C03648=1017.335,-79.595,386.221,-24.023,21.641,-43.975
C03649=1017.333,-79.935,386.245,-24.022,21.641,-43.981
C03650=1017.331,-80.274,386.270,-24.021,21.641,-43.986
C03651=1017.330,-80.613,386.294,-24.021,21.643,-43.990
C03652=1017.328,-80.952,386.319,-24.020,21.643,-43.995
C03653=1017.326,-81.290,386.344,-24.020,21.643,-44.001
C03654=1017.325,-81.627,386.368,-24.019,21.644,-44.005
C03655=1017.323,-81.965,386.392,-24.018,21.645,-44.010
C03656=1017.321,-82.302,386.417,-24.018,21.645,-44.016
C03657=1017.319,-82.639,386.441,-24.017,21.645,-44.021
C03658=1017.317,-82.974,386.465,-24.016,21.646,-44.025
C03659=1017.315,-83.310,386.490,-24.016,21.647,-44.031
C03660=1017.313,-83.646,386.514,-24.015,21.647,-44.036
C03661=1017.312,-83.981,386.538,-24.015,21.648,-44.040
C03662=1017.310,-84.315,386.562,-24.014,21.648,-44.045
C03663=1017.307,-84.664,386.587,-24.013,21.649,-44.051
C03664=1017.305,-85.062,386.616,-24.012,21.650,-44.056
C03665=1017.304,-85.273,386.631,-24.012,21.649,-44.060
C03666=1017.303,-85.488,386.647,-24.012,21.649,-44.062
C03667=1017.301,-85.897,386.676,-24.011,21.650,-44.067
C03668=1017.299,-86.255,386.702,-24.010,21.651,-44.073
C03669=1017.296,-86.585,386.726,-24.009,21.652,-44.078
C03670=1017.294,-86.907,386.749,-24.009,21.652,-44.082
C03671=1017.292,-87.224,386.772,-24.008,21.653,-44.088
C03672=1017.290,-87.536,386.794,-24.007,21.653,-44.093
C03673=1017.288,-87.847,386.816,-24.007,21.654,-44.097
C03674=1017.286,-88.160,386.839,-24.006,21.654,-44.102
C03675=1017.284,-88.478,386.861,-24.006,21.655,-44.106
C03676=1017.283,-88.849,386.888,-24.005,21.656,-44.114
C03677=1017.281,-89.068,386.904,-24.004,21.656,-44.117
C03678=1017.279,-89.302,386.921,-24.004,21.656,-44.119
C03679=1017.278,-89.540,386.938,-24.004,21.656,-44.121
C03680=1017.277,-89.771,386.954,-24.004,21.657,-44.123
C03681=1017.273,-90.177,386.983,-24.003,21.658,-44.130
C03682=1017.271,-90.516,387.008,-24.002,21.658,-44.136
C03683=1017.269,-90.845,387.031,-24.001,21.659,-44.141
C03684=1017.267,-91.173,387.055,-24.001,21.660,-44.145
C03685=1017.264,-91.502,387.078,-24.000,21.660,-44.150
C03686=1017.262,-91.831,387.101,-23.999,21.660,-44.156
C03687=1017.260,-92.159,387.125,-23.999,21.661,-44.160
C03688=1017.258,-92.486,387.148,-23.998,21.662,-44.165
C03689=1017.256,-92.813,387.171,-23.998,21.662,-44.169
C03690=1017.253,-93.139,387.194,-23.997,21.663,-44.175
C03691=1017.251,-93.465,387.218,-23.996,21.663,-44.180
C03692=1017.248,-93.789,387.240,-23.996,21.664,-44.184
C03693=1017.246,-94.114,387.264,-23.995,21.664,-44.189
C03694=1017.243,-94.438,387.287,-23.994,21.665,-44.193
C03695=1017.241,-94.762,387.310,-23.994,21.666,-44.199
C03696=1017.239,-95.085,387.333,-23.993,21.666,-44.204
C03697=1017.237,-95.407,387.356,-23.993,21.666,-44.207
C03698=1017.234,-95.729,387.378,-23.992,21.667,-44.213
C03699=1017.232,-96.052,387.402,-23.991,21.668,-44.217
C03700=1017.229,-96.373,387.424,-23.991,21.668,-44.222
C03701=1017.226,-96.695,387.447,-23.990,21.669,-44.226
C03702=1017.224,-97.016,387.469,-23.989,21.669,-44.231
C03703=1017.222,-97.337,387.492,-23.989,21.670,-44.236
C03704=1017.219,-97.658,387.515,-23.988,21.670,-44.241
C03705=1017.216,-97.979,387.538,-23.987,21.670,-44.246
C03706=1017.214,-98.300,387.560,-23.987,21.672,-44.250
C03707=1017.212,-98.620,387.583,-23.986,21.671,-44.255
C03708=1017.209,-98.942,387.605,-23.986,21.673,-44.260
C03709=1017.207,-99.263,387.628,-23.985,21.673,-44.265
C03710=1017.204,-99.585,387.651,-23.985,21.673,-44.268
C03711=1017.202,-99.906,387.673,-23.984,21.674,-44.274
C03712=1017.199,-100.227,387.696,-23.983,21.675,-44.278
C03713=1017.196,-100.551,387.719,-23.983,21.675,-44.283
C03714=1017.194,-100.872,387.742,-23.982,21.676,-44.287
C03715=1017.190,-101.196,387.764,-23.981,21.676,-44.292
C03716=1017.188,-101.519,387.786,-23.981,21.677,-44.298
C03717=1017.185,-101.843,387.810,-23.980,21.677,-44.302
C03718=1017.182,-102.168,387.833,-23.980,21.678,-44.307
C03719=1017.180,-102.493,387.855,-23.979,21.679,-44.311
C03720=1017.177,-102.818,387.878,-23.978,21.679,-44.316
C03721=1017.174,-103.145,387.901,-23.978,21.680,-44.320
C03722=1017.171,-103.471,387.924,-23.977,21.680,-44.326
C03723=1017.168,-103.798,387.947,-23.976,21.681,-44.331
C03724=1017.165,-104.125,387.970,-23.976,21.681,-44.335
C03725=1017.163,-104.453,387.992,-23.975,21.681,-44.340
C03726=1017.159,-104.781,388.016,-23.975,21.683,-44.344
C03727=1017.156,-105.110,388.038,-23.974,21.683,-44.350
C03728=1017.153,-105.438,388.061,-23.974,21.684,-44.354
C03729=1017.151,-105.767,388.084,-23.973,21.684,-44.359
C03730=1017.148,-106.096,388.107,-23.972,21.685,-44.365
C03731=1017.144,-106.425,388.130,-23.972,21.685,-44.368
C03732=1017.141,-106.754,388.153,-23.971,21.685,-44.374
C03733=1017.139,-107.083,388.176,-23.971,21.687,-44.378
C03734=1017.135,-107.412,388.199,-23.970,21.687,-44.383
C03735=1017.132,-107.740,388.222,-23.969,21.687,-44.388
C03736=1017.129,-108.070,388.245,-23.969,21.688,-44.392
C03737=1017.126,-108.398,388.268,-23.968,21.689,-44.398
C03738=1017.122,-108.727,388.291,-23.967,21.689,-44.402
C03739=1017.120,-109.056,388.314,-23.967,21.689,-44.407
C03740=1017.117,-109.385,388.337,-23.966,21.690,-44.412
C03741=1017.113,-109.714,388.360,-23.965,21.691,-44.416
C03742=1017.110,-110.043,388.382,-23.965,21.691,-44.422
C03743=1017.107,-110.372,388.404,-23.964,21.692,-44.426
C03744=1017.104,-110.701,388.427,-23.963,21.692,-44.431
C03745=1017.101,-111.030,388.450,-23.963,21.693,-44.436
C03746=1017.096,-111.359,388.473,-23.962,21.693,-44.440
C03747=1017.093,-111.687,388.495,-23.962,21.694,-44.446
C03748=1017.090,-112.016,388.518,-23.961,21.695,-44.449
C03749=1017.087,-112.345,388.541,-23.960,21.695,-44.455
C03750=1017.084,-112.674,388.564,-23.960,21.696,-44.459
C03751=1017.080,-113.002,388.587,-23.959,21.696,-44.464
C03752=1017.076,-113.330,388.609,-23.958,21.697,-44.470
C03753=1017.073,-113.659,388.632,-23.958,21.697,-44.473
C03754=1017.070,-113.988,388.655,-23.957,21.698,-44.479
C03755=1017.066,-114.316,388.677,-23.957,21.699,-44.483
C03756=1017.062,-114.645,388.700,-23.956,21.699,-44.488
C03757=1017.059,-114.974,388.723,-23.956,21.700,-44.492
C03758=1017.056,-115.302,388.745,-23.955,21.700,-44.497
C03759=1017.053,-115.631,388.768,-23.954,21.701,-44.503
C03760=1017.048,-115.960,388.790,-23.954,21.701,-44.507
C03761=1017.045,-116.288,388.813,-23.953,21.701,-44.512
C03762=1017.041,-116.616,388.836,-23.953,21.703,-44.516
C03763=1017.038,-116.945,388.858,-23.952,21.703,-44.521
C03764=1017.034,-117.273,388.881,-23.951,21.704,-44.525
C03765=1017.031,-117.602,388.904,-23.951,21.704,-44.531
C03766=1017.027,-117.930,388.926,-23.950,21.705,-44.535
C03767=1017.023,-118.259,388.948,-23.949,21.705,-44.540
C03768=1017.019,-118.588,388.971,-23.949,21.705,-44.545
C03769=1017.015,-118.915,388.994,-23.948,21.707,-44.549
C03770=1017.012,-119.244,389.016,-23.948,21.707,-44.554
C03771=1017.009,-119.572,389.038,-23.947,21.707,-44.558
C03772=1017.004,-119.901,389.061,-23.946,21.708,-44.564
C03773=1017.000,-120.229,389.083,-23.946,21.709,-44.568
C03774=1016.996,-120.557,389.106,-23.945,21.709,-44.573
C03775=1016.993,-120.885,389.128,-23.945,21.710,-44.577
C03776=1016.989,-121.214,389.150,-23.944,21.710,-44.582
C03777=1016.985,-121.543,389.173,-23.944,21.711,-44.586
C03778=1016.981,-121.871,389.196,-23.943,21.711,-44.591
C03779=1016.977,-122.199,389.218,-23.942,21.712,-44.597
C03780=1016.974,-122.510,389.239,-23.942,21.713,-44.601
C03781=1016.969,-122.856,389.263,-23.941,21.713,-44.606
C03782=1016.965,-123.184,389.285,-23.940,21.714,-44.610
C03783=1016.961,-123.512,389.308,-23.940,21.714,-44.615
C03784=1016.957,-123.840,389.330,-23.939,21.715,-44.620
C03785=1016.954,-124.168,389.352,-23.939,21.715,-44.625
C03786=1016.948,-124.496,389.374,-23.938,21.716,-44.628
C03787=1016.945,-124.825,389.396,-23.937,21.717,-44.634
C03788=1016.941,-125.153,389.419,-23.937,21.717,-44.638
C03789=1016.937,-125.481,389.441,-23.936,21.717,-44.643
C03790=1016.933,-125.809,389.463,-23.936,21.719,-44.647
C03791=1016.929,-126.138,389.486,-23.935,21.719,-44.652
C03792=1016.924,-126.466,389.507,-23.935,21.720,-44.657
C03793=1016.920,-126.793,389.530,-23.934,21.720,-44.662
C03794=1016.916,-127.122,389.552,-23.933,21.720,-44.667
C03795=1016.911,-127.450,389.574,-23.933,21.721,-44.671
C03796=1016.907,-127.778,389.597,-23.932,21.721,-44.676
C03797=1016.903,-128.106,389.619,-23.931,21.722,-44.680
C03798=1016.899,-128.434,389.641,-23.931,21.723,-44.686
C03799=1016.894,-128.762,389.664,-23.930,21.723,-44.689
C03800=1016.889,-129.090,389.685,-23.929,21.723,-44.695
C03801=1016.886,-129.419,389.707,-23.929,21.725,-44.699
C03802=1016.881,-129.746,389.730,-23.928,21.724,-44.704
C03803=1016.876,-130.075,389.752,-23.928,21.726,-44.708
C03804=1016.872,-130.403,389.774,-23.927,21.726,-44.713
C03805=1016.868,-130.730,389.796,-23.927,21.726,-44.717
C03806=1016.863,-131.058,389.818,-23.926,21.727,-44.723
C03807=1016.859,-131.387,389.840,-23.926,21.728,-44.726
C03808=1016.854,-131.715,389.863,-23.925,21.728,-44.732
C03809=1016.850,-132.043,389.884,-23.924,21.729,-44.736
C03810=1016.846,-132.370,389.907,-23.924,21.729,-44.741
C03811=1016.840,-132.699,389.929,-23.923,21.730,-44.745
C03812=1016.836,-133.027,389.950,-23.922,21.731,-44.750
C03813=1016.832,-133.354,389.973,-23.922,21.731,-44.754
C03814=1016.827,-133.683,389.995,-23.921,21.731,-44.759
C03815=1016.822,-134.010,390.017,-23.921,21.732,-44.763
C03816=1017.213,-133.983,389.773,-23.921,21.732,-44.763
C03817=1017.218,-133.655,389.751,-23.921,21.731,-44.759
C03818=1017.222,-133.327,389.730,-23.922,21.731,-44.754
C03819=1017.227,-132.998,389.706,-23.922,21.731,-44.750
C03820=1017.232,-132.670,389.685,-23.923,21.730,-44.745
C03821=1017.236,-132.342,389.663,-23.924,21.729,-44.741
C03822=1017.240,-132.014,389.641,-23.924,21.729,-44.736
C03823=1017.245,-131.687,389.619,-23.925,21.728,-44.732
C03824=1017.250,-131.358,389.597,-23.926,21.728,-44.726
C03825=1017.254,-131.030,389.575,-23.926,21.727,-44.723
C03826=1017.258,-130.703,389.553,-23.927,21.726,-44.717
C03827=1017.262,-130.374,389.531,-23.927,21.726,-44.713
C03828=1017.267,-130.047,389.509,-23.928,21.726,-44.708
C03829=1017.270,-129.718,389.487,-23.928,21.724,-44.704
C03830=1017.275,-129.391,389.465,-23.929,21.725,-44.699
C03831=1017.280,-129.062,389.442,-23.929,21.723,-44.695
C03832=1017.283,-128.734,389.420,-23.930,21.723,-44.689
C03833=1017.288,-128.406,389.399,-23.931,21.723,-44.686
C03834=1017.292,-128.078,389.376,-23.931,21.722,-44.680
C03835=1017.296,-127.750,389.354,-23.932,21.721,-44.676
C03836=1017.300,-127.422,389.332,-23.933,21.721,-44.671
C03837=1017.304,-127.094,389.310,-23.933,21.720,-44.667
C03838=1017.308,-126.766,389.287,-23.934,21.720,-44.662
C03839=1017.313,-126.437,389.265,-23.935,21.720,-44.657
C03840=1017.317,-126.109,389.243,-23.935,21.719,-44.652
C03841=1017.321,-125.781,389.221,-23.936,21.719,-44.647
C03842=1017.325,-125.453,389.199,-23.936,21.717,-44.643
C03843=1017.329,-125.125,389.176,-23.937,21.717,-44.638
C03844=1017.332,-124.797,389.154,-23.937,21.717,-44.634
C03845=1017.336,-124.469,389.132,-23.938,21.716,-44.628
C03846=1017.340,-124.140,389.110,-23.939,21.715,-44.625
C03847=1017.345,-123.812,389.088,-23.939,21.715,-44.620
C03848=1017.349,-123.484,389.065,-23.940,21.714,-44.615
C03849=1017.353,-123.156,389.043,-23.940,21.714,-44.610
C03850=1017.357,-122.828,389.021,-23.941,21.713,-44.606
C03851=1017.360,-122.499,388.999,-23.942,21.713,-44.601
C03852=1017.364,-122.171,388.976,-23.942,21.712,-44.597
C03853=1017.367,-121.842,388.954,-23.943,21.711,-44.591
C03854=1017.371,-121.515,388.932,-23.944,21.711,-44.586
C03855=1017.376,-121.186,388.909,-23.944,21.710,-44.582
C03856=1017.380,-120.858,388.887,-23.945,21.710,-44.577
C03857=1017.383,-120.529,388.865,-23.945,21.709,-44.573
C03858=1017.386,-120.201,388.842,-23.946,21.709,-44.568
C03859=1017.390,-119.873,388.820,-23.946,21.708,-44.564
C03860=1017.394,-119.544,388.798,-23.947,21.707,-44.558
C03861=1017.398,-119.217,388.775,-23.948,21.707,-44.554
C03862=1017.402,-118.887,388.752,-23.948,21.707,-44.549
C03863=1017.405,-118.559,388.730,-23.949,21.705,-44.545
C03864=1017.409,-118.231,388.708,-23.949,21.705,-44.540
C03865=1017.412,-117.902,388.685,-23.950,21.705,-44.535
C03866=1017.416,-117.574,388.663,-23.951,21.704,-44.531
C03867=1017.419,-117.245,388.640,-23.951,21.704,-44.525
C03868=1017.423,-116.917,388.618,-23.952,21.703,-44.521
C03869=1017.426,-116.588,388.595,-23.953,21.703,-44.516
C03870=1017.430,-116.260,388.573,-23.953,21.701,-44.512
C03871=1017.433,-115.931,388.550,-23.954,21.701,-44.507
C03872=1017.437,-115.603,388.528,-23.954,21.701,-44.503
C03873=1017.440,-115.275,388.505,-23.955,21.700,-44.497
C03874=1017.444,-114.947,388.483,-23.956,21.700,-44.492
C03875=1017.448,-114.617,388.460,-23.956,21.699,-44.488
C03876=1017.451,-114.289,388.437,-23.957,21.699,-44.483
C03877=1017.455,-113.961,388.415,-23.957,21.698,-44.479
C03878=1017.458,-113.632,388.392,-23.958,21.697,-44.473
C03879=1017.461,-113.303,388.369,-23.958,21.697,-44.470
C03880=1017.464,-112.974,388.347,-23.959,21.696,-44.464
C03881=1017.467,-112.646,388.324,-23.960,21.696,-44.459
C03882=1017.471,-112.317,388.302,-23.960,21.695,-44.455
C03883=1017.474,-111.989,388.279,-23.961,21.695,-44.449
C03884=1017.477,-111.659,388.257,-23.962,21.694,-44.446
C03885=1017.480,-111.330,388.234,-23.962,21.693,-44.440
C03886=1017.484,-111.002,388.211,-23.963,21.693,-44.436
C03887=1017.487,-110.672,388.188,-23.963,21.692,-44.431
C03888=1017.490,-110.344,388.166,-23.964,21.692,-44.426
C03889=1017.493,-110.015,388.143,-23.965,21.691,-44.422
C03890=1017.496,-109.687,388.120,-23.965,21.691,-44.416
C03891=1017.500,-109.357,388.097,-23.966,21.690,-44.412
C03892=1017.503,-109.029,388.074,-23.967,21.689,-44.407
C03893=1017.506,-108.700,388.052,-23.967,21.689,-44.402
C03894=1017.510,-108.371,388.029,-23.968,21.689,-44.398
C03895=1017.512,-108.042,388.006,-23.969,21.688,-44.392
C03896=1017.515,-107.713,387.983,-23.969,21.687,-44.388
C03897=1017.518,-107.384,387.960,-23.970,21.687,-44.383
C03898=1017.521,-107.055,387.938,-23.971,21.687,-44.378
C03899=1017.524,-106.725,387.914,-23.971,21.685,-44.374
C03900=1017.527,-106.397,387.891,-23.972,21.685,-44.368
C03901=1017.530,-106.068,387.869,-23.972,21.685,-44.365
C03902=1017.533,-105.739,387.847,-23.973,21.684,-44.359
C03903=1017.536,-105.410,387.823,-23.974,21.684,-44.354
C03904=1017.539,-105.082,387.800,-23.974,21.683,-44.350
C03905=1017.542,-104.754,387.777,-23.975,21.683,-44.344
C03906=1017.545,-104.425,387.754,-23.975,21.681,-44.340
C03907=1017.547,-104.098,387.731,-23.976,21.681,-44.335
C03908=1017.550,-103.771,387.708,-23.976,21.681,-44.331
C03909=1017.553,-103.444,387.685,-23.977,21.680,-44.326
C03910=1017.556,-103.117,387.663,-23.978,21.680,-44.320
C03911=1017.558,-102.791,387.640,-23.978,21.679,-44.316
C03912=1017.561,-102.466,387.617,-23.979,21.679,-44.311
C03913=1017.565,-102.140,387.594,-23.980,21.678,-44.307
C03914=1017.567,-101.815,387.572,-23.980,21.677,-44.302
C03915=1017.570,-101.492,387.549,-23.981,21.677,-44.298
C03916=1017.572,-101.168,387.526,-23.981,21.676,-44.292
C03917=1017.575,-100.845,387.504,-23.982,21.676,-44.287
C03918=1017.577,-100.522,387.481,-23.983,21.675,-44.283
C03919=1017.580,-100.200,387.459,-23.983,21.675,-44.278
C03920=1017.583,-99.878,387.436,-23.984,21.674,-44.274
C03921=1017.586,-99.557,387.413,-23.985,21.673,-44.268
C03922=1017.588,-99.235,387.391,-23.985,21.673,-44.265
C03923=1017.590,-98.914,387.369,-23.986,21.673,-44.260
C03924=1017.593,-98.593,387.345,-23.986,21.671,-44.255
C03925=1017.595,-98.272,387.323,-23.987,21.672,-44.250
C03926=1017.598,-97.951,387.300,-23.987,21.670,-44.246
C03927=1017.600,-97.631,387.277,-23.988,21.670,-44.241
C03928=1017.602,-97.310,387.255,-23.989,21.670,-44.236
C03929=1017.605,-96.988,387.232,-23.989,21.669,-44.231
C03930=1017.607,-96.667,387.210,-23.990,21.669,-44.226
C03931=1017.610,-96.347,387.187,-23.991,21.668,-44.222
C03932=1017.612,-96.025,387.164,-23.991,21.668,-44.217
C03933=1017.615,-95.703,387.141,-23.992,21.667,-44.213
C03934=1017.617,-95.381,387.118,-23.993,21.666,-44.207
C03935=1017.620,-95.057,387.096,-23.993,21.666,-44.204
C03936=1017.622,-94.735,387.073,-23.994,21.666,-44.199
C03937=1017.624,-94.412,387.050,-23.994,21.665,-44.193
C03938=1017.626,-94.086,387.027,-23.995,21.664,-44.189
C03939=1017.629,-93.762,387.004,-23.996,21.664,-44.184
C03940=1017.631,-93.437,386.981,-23.996,21.663,-44.180
C03941=1017.633,-93.111,386.958,-23.997,21.663,-44.175
C03942=1017.636,-92.785,386.934,-23.998,21.662,-44.169
C03943=1017.638,-92.459,386.911,-23.998,21.662,-44.165
C03944=1017.640,-92.131,386.888,-23.999,21.661,-44.160
C03945=1017.642,-91.804,386.864,-23.999,21.660,-44.156
C03946=1017.645,-91.475,386.841,-24.000,21.660,-44.150
C03947=1017.646,-91.147,386.818,-24.001,21.660,-44.145
C03948=1017.649,-90.817,386.794,-24.001,21.659,-44.141
C03949=1017.651,-90.488,386.771,-24.002,21.658,-44.136
C03950=1017.653,-90.150,386.746,-24.003,21.658,-44.130
C03951=1017.656,-89.744,386.718,-24.004,21.657,-44.123
C03952=1017.657,-89.513,386.701,-24.004,21.656,-44.121
C03953=1017.659,-89.275,386.684,-24.004,21.656,-44.119
C03954=1017.660,-89.041,386.667,-24.004,21.656,-44.117
C03955=1017.662,-88.822,386.652,-24.005,21.656,-44.114
C03956=1017.663,-88.451,386.625,-24.006,21.655,-44.106
C03957=1017.666,-88.132,386.602,-24.006,21.654,-44.102
C03958=1017.668,-87.819,386.580,-24.007,21.654,-44.097
C03959=1017.669,-87.509,386.557,-24.007,21.653,-44.093
C03960=1017.672,-87.196,386.536,-24.008,21.653,-44.088
C03961=1017.673,-86.880,386.513,-24.009,21.652,-44.082
C03962=1017.675,-86.558,386.490,-24.009,21.652,-44.078
C03963=1017.677,-86.228,386.466,-24.010,21.651,-44.073
C03964=1017.679,-85.869,386.440,-24.011,21.650,-44.067
C03965=1017.682,-85.460,386.411,-24.012,21.649,-44.062
C03966=1017.683,-85.246,386.395,-24.012,21.649,-44.060
C03967=1017.684,-85.034,386.380,-24.012,21.650,-44.056
C03968=1017.687,-84.637,386.351,-24.013,21.649,-44.051
C03969=1017.688,-84.287,386.326,-24.014,21.648,-44.045
C03970=1017.691,-83.953,386.302,-24.015,21.648,-44.040
C03971=1017.692,-83.618,386.278,-24.015,21.647,-44.036
C03972=1017.694,-83.283,386.254,-24.016,21.647,-44.031
C03973=1017.696,-82.947,386.230,-24.016,21.646,-44.025
C03974=1017.698,-82.611,386.206,-24.017,21.645,-44.021
C03975=1017.699,-82.275,386.181,-24.018,21.645,-44.016
C03976=1017.701,-81.938,386.157,-24.018,21.645,-44.010
C03977=1017.703,-81.600,386.132,-24.019,21.644,-44.005
C03978=1017.705,-81.262,386.108,-24.020,21.643,-44.001
C03979=1017.706,-80.925,386.083,-24.020,21.643,-43.995
C03980=1017.709,-80.586,386.058,-24.021,21.643,-43.990
C03981=1017.710,-80.247,386.034,-24.021,21.641,-43.986
C03982=1017.711,-79.907,386.010,-24.022,21.641,-43.981
C03983=1017.713,-79.568,385.985,-24.023,21.641,-43.975
C03984=1017.715,-79.227,385.960,-24.023,21.639,-43.971
C03985=1017.716,-78.886,385.935,-24.024,21.639,-43.966
C03986=1017.718,-78.546,385.910,-24.025,21.638,-43.960
C03987=1017.719,-78.205,385.886,-24.026,21.639,-43.955
C03988=1017.722,-77.863,385.861,-24.026,21.637,-43.951
C03989=1017.723,-77.522,385.836,-24.027,21.637,-43.946
C03990=1017.724,-77.180,385.811,-24.028,21.636,-43.940
C03991=1017.726,-76.837,385.786,-24.028,21.636,-43.936
C03992=1017.728,-76.495,385.761,-24.029,21.635,-43.931
C03993=1017.729,-76.152,385.736,-24.030,21.635,-43.926
C03994=1017.731,-75.809,385.711,-24.030,21.634,-43.920
C03995=1017.732,-75.467,385.686,-24.031,21.634,-43.916
C03996=1017.734,-75.123,385.660,-24.031,21.633,-43.911
C03997=1017.735,-74.780,385.635,-24.032,21.633,-43.905
C03998=1017.737,-74.436,385.611,-24.033,21.632,-43.901
C03999=1017.737,-74.093,385.585,-24.033,21.632,-43.896
C04000=1017.739,-73.749,385.560,-24.034,21.631,-43.890
C04001=1017.741,-73.405,385.534,-24.035,21.630,-43.885
C04002=1017.743,-73.062,385.509,-24.035,21.630,-43.881
C04003=1017.743,-72.718,385.485,-24.036,21.629,-43.875
C04004=1017.745,-72.374,385.459,-24.037,21.629,-43.870
C04005=1017.746,-72.030,385.434,-24.038,21.628,-43.865
C04006=1017.747,-71.686,385.409,-24.038,21.628,-43.861
C04007=1017.749,-71.342,385.383,-24.039,21.627,-43.855
C04008=1017.750,-70.997,385.358,-24.040,21.627,-43.850
C04009=1017.751,-70.653,385.333,-24.040,21.626,-43.844
C04010=1017.753,-70.309,385.307,-24.041,21.625,-43.840
C04011=1017.754,-69.965,385.282,-24.041,21.625,-43.835
C04012=1017.755,-69.621,385.257,-24.042,21.624,-43.829
C04013=1017.757,-69.277,385.231,-24.043,21.624,-43.824
C04014=1017.757,-68.933,385.206,-24.043,21.623,-43.820
C04015=1017.758,-68.589,385.180,-24.044,21.623,-43.815
C04016=1017.760,-68.246,385.155,-24.045,21.622,-43.809
C04017=1017.760,-67.902,385.129,-24.045,21.622,-43.805
C04018=1017.762,-67.559,385.104,-24.046,21.621,-43.800
C04019=1017.763,-67.215,385.079,-24.047,21.621,-43.795
C04020=1017.764,-66.872,385.053,-24.048,21.620,-43.789
C04021=1017.765,-66.530,385.028,-24.048,21.620,-43.785
C04022=1017.766,-66.187,385.002,-24.049,21.619,-43.780
C04023=1017.768,-65.844,384.977,-24.050,21.619,-43.774
C04024=1017.768,-65.501,384.951,-24.050,21.617,-43.770
C04025=1017.769,-65.160,384.926,-24.051,21.618,-43.765
C04026=1017.770,-64.818,384.901,-24.051,21.617,-43.759
C04027=1017.771,-64.476,384.875,-24.052,21.617,-43.754
C04028=1017.772,-64.135,384.849,-24.053,21.615,-43.750
C04029=1017.773,-63.794,384.824,-24.053,21.616,-43.745
C04030=1017.774,-63.453,384.799,-24.054,21.615,-43.739
C04031=1017.775,-63.113,384.773,-24.055,21.614,-43.735
C04032=1017.776,-62.773,384.748,-24.055,21.613,-43.730
C04033=1017.776,-62.433,384.723,-24.056,21.614,-43.725
C04034=1017.777,-62.095,384.697,-24.057,21.612,-43.720
C04035=1017.778,-61.756,384.672,-24.057,21.612,-43.715
C04036=1017.779,-61.417,384.646,-24.058,21.611,-43.710
C04037=1017.780,-61.079,384.621,-24.059,21.611,-43.706
C04038=1017.780,-60.742,384.597,-24.059,21.610,-43.700
C04039=1017.781,-60.404,384.571,-24.060,21.610,-43.695
C04040=1017.782,-60.067,384.545,-24.060,21.609,-43.691
C04041=1017.783,-59.731,384.520,-24.061,21.609,-43.686
C04042=1017.784,-59.394,384.495,-24.062,21.608,-43.680
C04043=1017.784,-59.059,384.470,-24.062,21.608,-43.676
C04044=1017.785,-58.724,384.445,-24.063,21.607,-43.671
C04045=1017.785,-58.389,384.420,-24.064,21.607,-43.666
C04046=1017.786,-58.054,384.395,-24.064,21.606,-43.662
C04047=1017.787,-57.720,384.369,-24.065,21.606,-43.656
C04048=1017.788,-57.386,384.345,-24.066,21.605,-43.652
C04049=1017.788,-57.053,384.319,-24.066,21.604,-43.647
C04050=1017.789,-56.719,384.294,-24.067,21.605,-43.642
C04051=1017.788,-56.386,384.269,-24.068,21.603,-43.637
C04052=1017.790,-56.053,384.244,-24.068,21.603,-43.632
C04053=1017.790,-55.721,384.218,-24.069,21.603,-43.627
C04054=1017.790,-55.387,384.193,-24.070,21.602,-43.623
C04055=1017.791,-55.055,384.168,-24.070,21.602,-43.618
C04056=1017.791,-54.722,384.143,-24.071,21.601,-43.613
C04057=1017.792,-54.391,384.118,-24.072,21.601,-43.608
C04058=1017.792,-54.058,384.093,-24.072,21.600,-43.603
C04059=1017.793,-53.726,384.068,-24.073,21.599,-43.599
C04060=1017.793,-53.394,384.042,-24.074,21.600,-43.594
C04061=1017.794,-53.061,384.018,-24.074,21.598,-43.589
C04062=1017.794,-52.729,383.992,-24.075,21.598,-43.584
C04063=1017.795,-52.397,383.966,-24.075,21.597,-43.579
C04064=1017.795,-52.064,383.942,-24.076,21.597,-43.575
C04065=1017.795,-51.732,383.916,-24.077,21.597,-43.570
C04066=1017.796,-51.400,383.891,-24.077,21.596,-43.566
C04067=1017.796,-51.067,383.866,-24.078,21.596,-43.560
C04068=1017.797,-50.735,383.841,-24.079,21.595,-43.555
C04069=1017.797,-50.403,383.815,-24.079,21.594,-43.551
C04070=1017.797,-50.070,383.790,-24.080,21.595,-43.546
C04071=1017.797,-49.738,383.764,-24.080,21.593,-43.542
C04072=1017.797,-49.405,383.739,-24.081,21.593,-43.536
C04073=1017.798,-49.073,383.714,-24.081,21.592,-43.532
C04074=1017.798,-48.741,383.689,-24.082,21.592,-43.527
C04075=1017.798,-48.408,383.664,-24.083,21.592,-43.522
C04076=1017.798,-48.076,383.638,-24.083,21.591,-43.518
C04077=1017.799,-47.742,383.613,-24.084,21.591,-43.512
C04078=1017.799,-47.410,383.587,-24.085,21.589,-43.508
C04079=1017.799,-47.078,383.561,-24.086,21.589,-43.503
C04080=1017.799,-46.745,383.536,-24.086,21.590,-43.498
C04081=1017.799,-46.413,383.510,-24.087,21.588,-43.494
C04082=1017.800,-46.081,383.485,-24.088,21.588,-43.488
C04083=1017.800,-45.748,383.460,-24.088,21.588,-43.485
C04084=1017.800,-45.416,383.434,-24.089,21.587,-43.479
C04085=1017.799,-45.083,383.409,-24.089,21.586,-43.475
C04086=1017.799,-44.750,383.383,-24.090,21.586,-43.470
C04087=1017.799,-44.418,383.357,-24.091,21.586,-43.465
C04088=1017.799,-44.085,383.332,-24.091,21.585,-43.461
C04089=1017.800,-43.753,383.306,-24.092,21.585,-43.455
C04090=1017.800,-43.420,383.280,-24.092,21.584,-43.451
C04091=1017.800,-43.087,383.255,-24.093,21.583,-43.446
C04092=1017.800,-42.755,383.229,-24.094,21.583,-43.442
C04093=1017.800,-42.422,383.204,-24.094,21.583,-43.437
C04094=1017.799,-42.090,383.178,-24.095,21.582,-43.431
C04095=1017.799,-41.757,383.152,-24.096,21.582,-43.427
C04096=1017.799,-41.425,383.127,-24.096,21.582,-43.422
C04097=1017.799,-41.092,383.101,-24.097,21.580,-43.418
C04098=1017.799,-40.760,383.075,-24.098,21.580,-43.413
C04099=1017.798,-40.427,383.050,-24.098,21.580,-43.409
C04100=1017.798,-40.095,383.024,-24.099,21.579,-43.404
C04101=1017.799,-39.761,382.997,-24.100,21.579,-43.398
C04102=1017.798,-39.429,382.972,-24.100,21.578,-43.394
C04103=1017.798,-39.096,382.946,-24.101,21.578,-43.389
C04104=1017.798,-38.764,382.920,-24.101,21.577,-43.385
C04105=1017.797,-38.431,382.895,-24.102,21.577,-43.380
C04106=1017.798,-38.098,382.869,-24.102,21.576,-43.376
C04107=1017.797,-37.766,382.843,-24.103,21.576,-43.371
C04108=1017.797,-37.433,382.818,-24.104,21.575,-43.366
C04109=1017.797,-37.101,382.792,-24.105,21.575,-43.361
C04110=1017.796,-36.768,382.765,-24.105,21.574,-43.357
C04111=1017.796,-36.435,382.740,-24.106,21.574,-43.352
C04112=1017.795,-36.103,382.714,-24.107,21.574,-43.347
C04113=1017.796,-35.770,382.687,-24.107,21.573,-43.343
C04114=1017.795,-35.436,382.662,-24.108,21.573,-43.337
C04115=1017.795,-35.104,382.636,-24.108,21.572,-43.334
C04116=1017.794,-34.772,382.610,-24.109,21.572,-43.328
C04117=1017.794,-34.439,382.584,-24.109,21.571,-43.324
C04118=1017.793,-34.106,382.558,-24.110,21.571,-43.319
C04119=1017.793,-33.774,382.532,-24.111,21.570,-43.315
C04120=1017.793,-33.441,382.506,-24.111,21.570,-43.310
C04121=1017.792,-33.108,382.481,-24.112,21.569,-43.306
C04122=1017.791,-32.776,382.454,-24.113,21.569,-43.301
C04123=1017.791,-32.443,382.428,-24.113,21.568,-43.296
C04124=1017.790,-32.110,382.402,-24.114,21.568,-43.291
C04125=1017.790,-31.777,382.376,-24.114,21.567,-43.287
C04126=1017.790,-31.444,382.349,-24.115,21.567,-43.282
C04127=1017.789,-31.112,382.323,-24.116,21.566,-43.278
C04128=1017.788,-30.779,382.298,-24.116,21.566,-43.273
C04129=1017.788,-30.446,382.271,-24.117,21.565,-43.269
C04130=1017.787,-30.114,382.245,-24.118,21.565,-43.264
C04131=1017.787,-29.781,382.219,-24.118,21.565,-43.260
C04132=1017.786,-29.448,382.193,-24.119,21.564,-43.254
C04133=1017.786,-29.115,382.167,-24.119,21.563,-43.250
C04134=1017.785,-28.783,382.141,-24.120,21.563,-43.245
C04135=1017.784,-28.450,382.115,-24.120,21.562,-43.241
C04136=1017.783,-28.117,382.088,-24.121,21.562,-43.236
C04137=1017.782,-27.784,382.062,-24.122,21.562,-43.232
C04138=1017.782,-27.452,382.036,-24.123,21.562,-43.227
C04139=1017.781,-27.119,382.009,-24.123,21.560,-43.223
C04140=1017.781,-26.786,381.984,-24.124,21.560,-43.217
C04141=1017.779,-26.453,381.957,-24.124,21.560,-43.214
C04142=1017.779,-26.121,381.931,-24.125,21.559,-43.208
C04143=1017.778,-25.788,381.904,-24.126,21.559,-43.204
C04144=1017.778,-25.455,381.879,-24.126,21.559,-43.199
C04145=1017.777,-25.122,381.852,-24.127,21.558,-43.195
C04146=1017.776,-24.789,381.825,-24.128,21.558,-43.190
C04147=1017.776,-24.457,381.799,-24.128,21.557,-43.186
C04148=1017.775,-24.124,381.772,-24.129,21.557,-43.181
C04149=1017.774,-23.791,381.746,-24.129,21.556,-43.177
C04150=1017.773,-23.458,381.720,-24.130,21.556,-43.171
C04151=1017.772,-23.125,381.693,-24.131,21.555,-43.168
C04152=1017.771,-22.793,381.666,-24.131,21.556,-43.162
C04153=1017.770,-22.460,381.640,-24.132,21.554,-43.158
C04154=1017.769,-22.127,381.614,-24.133,21.554,-43.153
C04155=1017.768,-21.794,381.588,-24.133,21.554,-43.149
C04156=1017.767,-21.461,381.561,-24.134,21.553,-43.144
C04157=1017.766,-21.129,381.535,-24.134,21.552,-43.140
C04158=1017.765,-20.796,381.508,-24.135,21.553,-43.135
C04159=1017.764,-20.463,381.482,-24.136,21.552,-43.131
C04160=1017.763,-20.130,381.455,-24.136,21.551,-43.127
C04161=1017.762,-19.797,381.428,-24.137,21.551,-43.122
C04162=1017.762,-19.626,381.415,-24.137,21.550,-43.118
C04163=1017.760,-19.209,381.381,-24.138,21.550,-43.112
C04164=1017.760,-18.961,381.362,-24.139,21.550,-43.109
C04165=1017.759,-18.699,381.341,-24.139,21.550,-43.107
C04166=1017.758,-18.437,381.320,-24.139,21.549,-43.105
C04167=1017.757,-18.190,381.300,-24.139,21.548,-43.103
C04168=1017.757,-17.968,381.283,-24.140,21.549,-43.100
C04169=1017.755,-17.603,381.253,-24.141,21.548,-43.092
C04170=1017.754,-17.270,381.227,-24.141,21.547,-43.088
C04171=1017.753,-16.937,381.200,-24.142,21.547,-43.083
C04172=1017.751,-16.604,381.173,-24.142,21.547,-43.079
C04173=1017.750,-16.270,381.146,-24.143,21.546,-43.074
C04174=1017.749,-15.936,381.120,-24.144,21.546,-43.070
C04175=1017.748,-15.601,381.093,-24.145,21.546,-43.065
C04176=1017.747,-15.265,381.065,-24.145,21.545,-43.061
C04177=1017.745,-14.926,381.039,-24.146,21.544,-43.055
C04178=1017.744,-14.586,381.012,-24.146,21.544,-43.052
C04179=1017.743,-14.244,380.984,-24.147,21.544,-43.046
C04180=1017.741,-13.900,380.956,-24.147,21.543,-43.042
C04181=1017.740,-13.554,380.928,-24.148,21.543,-43.037
C04182=1017.739,-13.205,380.901,-24.149,21.542,-43.033
C04183=1017.737,-12.855,380.872,-24.149,21.542,-43.028
C04184=1017.736,-12.504,380.843,-24.150,21.541,-43.024
C04185=1017.735,-12.150,380.815,-24.151,21.541,-43.019
C04186=1017.733,-11.794,380.786,-24.151,21.540,-43.014
C04187=1017.732,-11.438,380.758,-24.152,21.540,-43.009
C04188=1017.730,-11.080,380.729,-24.152,21.539,-43.006
C04189=1017.729,-10.721,380.700,-24.153,21.539,-43.000
C04190=1017.728,-10.362,380.671,-24.154,21.539,-42.995
C04191=1017.725,-10.001,380.641,-24.154,21.538,-42.991
C04192=1017.723,-9.639,380.612,-24.155,21.538,-42.985
C04193=1017.722,-9.277,380.583,-24.156,21.537,-42.982
C04194=1017.721,-8.914,380.554,-24.156,21.536,-42.976
C04195=1017.719,-8.551,380.524,-24.157,21.536,-42.971
C04196=1017.718,-8.189,380.495,-24.158,21.536,-42.967
C04197=1017.716,-7.826,380.465,-24.158,21.535,-42.961
C04198=1017.715,-7.459,380.436,-24.159,21.535,-42.956
C04199=1017.712,-7.090,380.406,-24.160,21.534,-42.952
C04200=1017.711,-6.719,380.376,-24.160,21.534,-42.947
C04201=1017.709,-6.344,380.345,-24.161,21.533,-42.941
C04202=1017.707,-5.969,380.315,-24.162,21.533,-42.937
C04203=1017.705,-5.593,380.285,-24.163,21.533,-42.932
C04204=1017.703,-5.219,380.254,-24.163,21.532,-42.928
C04205=1017.702,-4.849,380.223,-24.164,21.532,-42.923
C04206=1017.700,-4.483,380.194,-24.164,21.531,-42.919
C04207=1017.697,-4.121,380.165,-24.165,21.530,-42.913
C04208=1017.696,-3.765,380.135,-24.166,21.531,-42.908
C04209=1017.695,-3.410,380.107,-24.166,21.529,-42.904
C04210=1017.692,-3.057,380.078,-24.167,21.529,-42.899
C04211=1017.691,-2.706,380.048,-24.167,21.529,-42.895
C04212=1017.689,-2.356,380.021,-24.168,21.529,-42.890
C04213=1017.686,-2.008,379.992,-24.169,21.528,-42.886
C04214=1017.685,-1.661,379.964,-24.169,21.528,-42.880
C04215=1017.683,-1.316,379.936,-24.170,21.527,-42.877
C04216=1017.681,-0.972,379.907,-24.170,21.527,-42.873
C04217=1017.679,-0.631,379.879,-24.171,21.526,-42.867
C04218=1017.677,-0.291,379.852,-24.172,21.526,-42.864
C04219=1017.675,0.048,379.824,-24.172,21.526,-42.858
C04220=1017.674,0.384,379.796,-24.173,21.525,-42.855
C04221=1017.672,0.721,379.769,-24.173,21.525,-42.851
C04222=1017.669,1.055,379.741,-24.174,21.525,-42.846
C04223=1017.668,1.389,379.713,-24.175,21.524,-42.842
C04224=1017.666,1.723,379.687,-24.175,21.523,-42.838
C04225=1017.664,2.053,379.659,-24.176,21.523,-42.834
C04226=1017.662,2.366,379.633,-24.176,21.523,-42.831
C04227=1017.661,2.654,379.610,-24.177,21.522,-42.827
C04228=1017.659,2.922,379.588,-24.177,21.522,-42.823
C04229=1017.657,3.185,379.567,-24.178,21.522,-42.818
C04230=1017.655,3.454,379.544,-24.179,21.521,-42.814
C04231=1017.654,3.743,379.520,-24.179,21.521,-42.810
C04232=1017.652,4.056,379.495,-24.179,21.520,-42.807
C04233=1017.650,4.387,379.467,-24.180,21.521,-42.803
C04234=1017.648,4.717,379.440,-24.180,21.519,-42.799
C04235=1017.646,5.049,379.412,-24.181,21.519,-42.795
C04236=1017.644,5.380,379.385,-24.181,21.518,-42.792
C04237=1017.642,5.710,379.358,-24.182,21.519,-42.786
C04238=1017.639,6.040,379.331,-24.183,21.518,-42.783
C04239=1017.638,6.369,379.304,-24.183,21.518,-42.779
C04240=1017.635,6.698,379.277,-24.184,21.518,-42.774
C04241=1017.634,7.027,379.250,-24.185,21.517,-42.770
C04242=1017.631,7.355,379.222,-24.185,21.517,-42.766
C04243=1017.629,7.680,379.196,-24.186,21.516,-42.762
C04244=1017.627,8.003,379.169,-24.186,21.516,-42.759
C04245=1017.625,8.324,379.142,-24.186,21.515,-42.755
C04246=1017.623,8.642,379.115,-24.187,21.516,-42.750
C04247=1017.621,8.959,379.090,-24.188,21.515,-42.746
C04248=1017.619,9.273,379.064,-24.188,21.515,-42.742
C04249=1017.616,9.588,379.038,-24.189,21.514,-42.738
C04250=1017.614,9.903,379.012,-24.190,21.514,-42.733
C04251=1017.612,10.219,378.986,-24.190,21.514,-42.730
C04252=1017.610,10.536,378.958,-24.191,21.513,-42.726
C04253=1017.607,10.854,378.932,-24.191,21.513,-42.722
C04254=1017.605,11.175,378.906,-24.192,21.512,-42.718
C04255=1017.603,11.497,378.879,-24.192,21.512,-42.715
C04256=1017.601,11.820,378.852,-24.193,21.511,-42.711
C04257=1017.599,12.144,378.825,-24.193,21.511,-42.707
C04258=1017.596,12.467,378.799,-24.194,21.511,-42.702
C04259=1017.594,12.791,378.771,-24.194,21.510,-42.698
C04260=1017.591,13.115,378.745,-24.195,21.510,-42.694
C04261=1017.589,13.439,378.718,-24.195,21.509,-42.691
C04262=1017.587,13.762,378.690,-24.196,21.509,-42.687
C04263=1017.584,14.086,378.664,-24.197,21.509,-42.682
C04264=1017.582,14.411,378.636,-24.197,21.509,-42.678
C04265=1017.580,14.737,378.610,-24.198,21.508,-42.674
C04266=1017.577,15.062,378.582,-24.198,21.508,-42.670
C04267=1017.574,15.388,378.555,-24.199,21.507,-42.667
C04268=1017.572,15.714,378.528,-24.199,21.507,-42.663
C04269=1017.569,16.041,378.501,-24.200,21.507,-42.658
C04270=1017.567,16.369,378.473,-24.200,21.506,-42.654
C04271=1017.564,16.697,378.445,-24.201,21.506,-42.650
C04272=1017.562,17.026,378.418,-24.201,21.505,-42.646
C04273=1017.559,17.354,378.391,-24.202,21.505,-42.643
C04274=1017.557,17.684,378.363,-24.202,21.504,-42.639
C04275=1017.554,18.015,378.336,-24.203,21.504,-42.634
C04276=1017.551,18.345,378.308,-24.204,21.504,-42.630
C04277=1017.549,18.677,378.280,-24.204,21.503,-42.626
C04278=1017.547,19.009,378.252,-24.205,21.503,-42.622
C04279=1017.543,19.342,378.224,-24.205,21.502,-42.619
C04280=1017.541,19.689,378.195,-24.206,21.503,-42.613
C04281=1017.537,20.106,378.161,-24.207,21.502,-42.608
C04282=1017.535,20.342,378.140,-24.207,21.502,-42.604
C04283=1017.534,20.589,378.120,-24.207,21.502,-42.603
C04284=1017.531,20.837,378.099,-24.208,21.502,-42.601
C04285=1017.530,21.079,378.079,-24.208,21.502,-42.599
C04286=1017.527,21.306,378.060,-24.208,21.501,-42.597
C04287=1017.526,21.514,378.042,-24.209,21.501,-42.593
C04288=1017.523,21.870,378.012,-24.209,21.500,-42.588
C04289=1017.520,22.194,377.985,-24.210,21.501,-42.584
C04290=1017.518,22.488,377.960,-24.210,21.500,-42.582
C04291=1017.515,22.742,377.939,-24.210,21.499,-42.580
C04292=1017.512,23.151,377.905,-24.211,21.499,-42.573
C04293=1017.508,23.558,377.870,-24.212,21.498,-42.565
C04294=1017.506,23.811,377.849,-24.213,21.498,-42.562
C04295=1017.504,24.105,377.825,-24.213,21.498,-42.560
C04296=1017.501,24.432,377.797,-24.213,21.497,-42.558
C04297=1017.498,24.766,377.769,-24.214,21.497,-42.553
C04298=1017.495,25.100,377.740,-24.215,21.497,-42.549
C04299=1017.492,25.435,377.713,-24.215,21.496,-42.545
C04300=1017.489,25.769,377.684,-24.216,21.496,-42.541
C04301=1017.487,26.104,377.656,-24.216,21.495,-42.538
C04302=1017.483,26.437,377.628,-24.217,21.495,-42.534
C04303=1017.480,26.772,377.599,-24.217,21.494,-42.530
C04304=1017.477,27.106,377.571,-24.218,21.494,-42.525
C04305=1017.474,27.441,377.543,-24.219,21.495,-42.522
C04306=1017.471,27.775,377.515,-24.219,21.494,-42.518
C04307=1017.468,28.110,377.487,-24.220,21.494,-42.514
C04308=1017.465,28.443,377.458,-24.220,21.493,-42.510
C04309=1017.462,28.778,377.430,-24.221,21.493,-42.507
C04310=1017.459,29.113,377.401,-24.221,21.492,-42.503
C04311=1017.456,29.447,377.373,-24.222,21.493,-42.498
C04312=1017.453,29.782,377.344,-24.222,21.492,-42.494
C04313=1017.449,30.116,377.316,-24.223,21.492,-42.490
C04314=1017.446,30.451,377.289,-24.223,21.491,-42.486
C04315=1017.443,30.785,377.260,-24.224,21.491,-42.483
C04316=1017.440,31.120,377.232,-24.224,21.490,-42.479
C04317=1017.436,31.453,377.203,-24.225,21.490,-42.475
C04318=1017.433,31.789,377.175,-24.225,21.489,-42.471
C04319=1017.430,32.124,377.146,-24.226,21.489,-42.468
C04320=1017.427,32.457,377.118,-24.226,21.489,-42.464
C04321=1017.423,32.793,377.089,-24.227,21.489,-42.459
C04322=1017.420,33.126,377.061,-24.228,21.489,-42.455
C04323=1017.417,33.461,377.032,-24.228,21.488,-42.452
C04324=1017.414,33.797,377.004,-24.229,21.488,-42.448
C04325=1017.410,34.130,376.975,-24.229,21.487,-42.444
C04326=1017.407,34.465,376.947,-24.230,21.487,-42.440
C04327=1017.403,34.800,376.919,-24.230,21.486,-42.437
C04328=1017.400,35.134,376.890,-24.231,21.486,-42.433
C04329=1017.397,35.470,376.862,-24.231,21.485,-42.429
C04330=1017.394,35.803,376.833,-24.232,21.486,-42.426
C04331=1017.390,36.138,376.805,-24.232,21.485,-42.422
C04332=1017.387,36.474,376.776,-24.233,21.485,-42.418
C04333=1017.383,36.808,376.747,-24.234,21.485,-42.413
C04334=1017.380,37.143,376.719,-24.234,21.485,-42.409
C04335=1017.376,37.477,376.691,-24.235,21.484,-42.405
C04336=1017.373,37.812,376.661,-24.235,21.484,-42.402
C04337=1017.369,38.147,376.633,-24.236,21.483,-42.398
C04338=1017.366,38.481,376.605,-24.236,21.483,-42.395
C04339=1017.363,38.816,376.576,-24.237,21.483,-42.391
C04340=1017.359,39.151,376.547,-24.237,21.483,-42.387
C04341=1017.355,39.486,376.519,-24.238,21.482,-42.383
C04342=1017.351,39.821,376.490,-24.238,21.482,-42.380
C04343=1017.348,40.155,376.462,-24.239,21.481,-42.376
C04344=1017.344,40.490,376.433,-24.239,21.481,-42.372
C04345=1017.341,40.826,376.404,-24.240,21.481,-42.369
C04346=1017.337,41.159,376.376,-24.240,21.481,-42.365
C04347=1017.333,41.495,376.347,-24.241,21.480,-42.361
C04348=1017.330,41.830,376.318,-24.241,21.480,-42.357
C04349=1017.325,42.165,376.290,-24.242,21.479,-42.354
C04350=1017.323,42.499,376.261,-24.242,21.479,-42.350
C04351=1017.318,42.834,376.232,-24.243,21.479,-42.347
C04352=1017.315,43.169,376.204,-24.243,21.479,-42.343
C04353=1017.311,43.504,376.174,-24.244,21.478,-42.339
C04354=1017.307,43.838,376.146,-24.244,21.478,-42.335
C04355=1017.304,44.174,376.118,-24.245,21.477,-42.332
C04356=1017.300,44.509,376.089,-24.245,21.477,-42.328
C04357=1017.295,44.843,376.059,-24.246,21.477,-42.325
C04358=1017.292,45.178,376.031,-24.246,21.477,-42.321
C04359=1017.288,45.513,376.003,-24.247,21.476,-42.317
C04360=1017.284,45.848,375.974,-24.247,21.476,-42.313
C04361=1017.281,46.183,375.945,-24.248,21.475,-42.309
C04362=1017.277,46.518,375.916,-24.248,21.475,-42.306
C04363=1017.273,46.853,375.887,-24.249,21.475,-42.302
C04364=1017.268,47.188,375.859,-24.249,21.475,-42.299
C04365=1017.264,47.523,375.829,-24.250,21.474,-42.295
C04366=1017.261,47.858,375.801,-24.250,21.474,-42.291
C04367=1017.257,48.192,375.772,-24.251,21.473,-42.287
C04368=1017.253,48.528,375.743,-24.251,21.473,-42.284
C04369=1017.249,48.862,375.714,-24.252,21.473,-42.280
C04370=1017.245,49.197,375.685,-24.252,21.473,-42.277
C04371=1017.241,49.533,375.656,-24.253,21.472,-42.273
C04372=1017.236,49.867,375.628,-24.253,21.472,-42.269
C04373=1017.233,50.202,375.598,-24.254,21.472,-42.266
C04374=1017.228,50.537,375.569,-24.254,21.471,-42.262
C04375=1017.224,50.872,375.540,-24.255,21.471,-42.258
C04376=1017.220,51.207,375.512,-24.255,21.471,-42.254
C04377=1017.216,51.542,375.482,-24.256,21.471,-42.251
C04378=1017.212,51.877,375.453,-24.256,21.470,-42.247
C04379=1017.208,52.212,375.425,-24.257,21.470,-42.244
C04380=1017.204,52.548,375.396,-24.257,21.470,-42.240
C04381=1017.200,52.882,375.367,-24.258,21.469,-42.238
C04382=1017.196,53.217,375.338,-24.258,21.469,-42.234
C04383=1017.191,53.552,375.309,-24.259,21.468,-42.230
C04384=1017.187,53.887,375.280,-24.259,21.468,-42.227
C04385=1017.183,54.222,375.252,-24.260,21.468,-42.223
C04386=1017.179,54.557,375.222,-24.260,21.468,-42.220
C04387=1017.174,54.892,375.193,-24.261,21.467,-42.216
C04388=1017.170,55.227,375.164,-24.261,21.467,-42.212
C04389=1017.165,55.562,375.136,-24.262,21.467,-42.209
C04390=1017.162,55.897,375.106,-24.262,21.467,-42.205
C04391=1017.157,56.231,375.077,-24.263,21.466,-42.201
C04392=1017.153,56.567,375.048,-24.263,21.466,-42.197
C04393=1017.148,56.902,375.019,-24.264,21.466,-42.194
C04394=1017.144,57.237,374.990,-24.264,21.465,-42.192
C04395=1017.139,57.572,374.961,-24.264,21.465,-42.188
C04396=1017.135,57.907,374.932,-24.265,21.464,-42.184
C04397=1017.131,58.242,374.903,-24.266,21.465,-42.181
C04398=1017.126,58.577,374.874,-24.266,21.464,-42.177
C04399=1017.122,58.912,374.844,-24.267,21.464,-42.173
C04400=1017.118,59.246,374.816,-24.267,21.464,-42.170
C04401=1017.113,59.582,374.786,-24.268,21.464,-42.166
C04402=1017.108,59.917,374.758,-24.268,21.463,-42.163
C04403=1017.105,60.252,374.728,-24.268,21.462,-42.160
C04404=1017.099,60.587,374.699,-24.269,21.462,-42.157
C04405=1017.095,60.922,374.670,-24.269,21.462,-42.153
C04406=1017.090,61.257,374.641,-24.270,21.461,-42.149
C04407=1017.086,61.592,374.612,-24.270,21.462,-42.146
C04408=1017.081,61.926,374.583,-24.271,21.461,-42.142
C04409=1017.077,62.262,374.554,-24.271,21.461,-42.139
C04410=1017.072,62.598,374.525,-24.272,21.460,-42.135
C04411=1017.066,62.994,374.490,-24.272,21.460,-42.131
C04412=1017.063,63.218,374.470,-24.273,21.461,-42.130
C04413=1017.060,63.436,374.452,-24.273,21.460,-42.128
C04414=1017.058,63.810,374.417,-24.274,21.460,-42.124
C04415=1017.057,64.166,374.383,-24.274,21.459,-42.120
C04416=1017.057,64.552,374.347,-24.274,21.459,-42.116
C04417=1017.055,64.947,374.310,-24.275,21.458,-42.113
C04418=1017.054,65.325,374.274,-24.276,21.459,-42.108
C04419=1017.053,65.680,374.241,-24.276,21.457,-42.105
C04420=1017.052,66.018,374.209,-24.277,21.458,-42.102
C04421=1017.051,66.351,374.178,-24.277,21.457,-42.098
C04422=1017.051,66.687,374.146,-24.278,21.457,-42.094
C04423=1017.050,67.024,374.114,-24.278,21.457,-42.091
C04424=1017.048,67.361,374.082,-24.279,21.457,-42.087
C04425=1017.047,67.699,374.050,-24.279,21.456,-42.085
C04426=1017.046,68.038,374.018,-24.279,21.456,-42.082
C04427=1017.046,68.379,373.986,-24.280,21.456,-42.078
C04428=1017.044,68.720,373.954,-24.280,21.455,-42.074
C04429=1017.044,69.062,373.921,-24.281,21.456,-42.071
C04430=1017.043,69.405,373.889,-24.281,21.455,-42.067
C04431=1017.041,69.749,373.856,-24.282,21.455,-42.063
C04432=1017.041,70.093,373.824,-24.282,21.454,-42.061
C04433=1017.039,70.437,373.791,-24.283,21.454,-42.058
C04434=1017.038,70.782,373.758,-24.283,21.453,-42.054
C04435=1017.037,71.126,373.725,-24.284,21.454,-42.051
C04436=1017.036,71.471,373.693,-24.284,21.453,-42.047
C04437=1017.035,71.816,373.660,-24.285,21.453,-42.043
C04438=1017.034,72.161,373.627,-24.285,21.453,-42.041
C04439=1017.033,72.508,373.595,-24.285,21.452,-42.037
C04440=1017.031,72.856,373.561,-24.286,21.452,-42.034
C04441=1017.032,73.205,373.528,-24.286,21.451,-42.030
C04442=1017.030,73.556,373.495,-24.287,21.452,-42.027
C04443=1017.028,73.910,373.461,-24.288,21.451,-42.023
C04444=1017.027,74.265,373.427,-24.288,21.451,-42.019
C04445=1017.027,74.622,373.393,-24.288,21.451,-42.017
C04446=1017.025,74.981,373.359,-24.289,21.450,-42.013
C04447=1017.025,75.338,373.325,-24.289,21.450,-42.010
C04448=1017.023,75.691,373.291,-24.290,21.450,-42.006
C04449=1017.022,76.041,373.258,-24.290,21.449,-42.004
C04450=1017.021,76.382,373.225,-24.291,21.449,-42.001
C04451=1017.020,76.719,373.194,-24.291,21.449,-41.997
C04452=1017.018,77.049,373.162,-24.292,21.449,-41.994
C04453=1017.018,77.375,373.130,-24.292,21.449,-41.990
C04454=1017.016,77.699,373.100,-24.292,21.448,-41.987
C04455=1017.015,78.022,373.069,-24.293,21.448,-41.984
C04456=1017.014,78.346,373.037,-24.293,21.448,-41.980
C04457=1017.013,78.674,373.006,-24.294,21.447,-41.977
C04458=1017.013,79.007,372.974,-24.295,21.448,-41.973
C04459=1017.011,79.347,372.941,-24.295,21.446,-41.971
C04460=1017.011,79.691,372.908,-24.295,21.447,-41.968
C04461=1017.009,80.042,372.875,-24.296,21.446,-41.964
C04462=1017.008,80.398,372.841,-24.296,21.446,-41.962
C04463=1017.007,80.754,372.806,-24.297,21.446,-41.958
C04464=1017.005,81.111,372.772,-24.297,21.445,-41.955
C04465=1017.005,81.466,372.738,-24.298,21.446,-41.951
C04466=1017.003,81.822,372.704,-24.298,21.445,-41.947
C04467=1017.002,82.176,372.669,-24.298,21.444,-41.945
C04468=1017.002,82.530,372.636,-24.299,21.444,-41.942
C04469=1017.000,82.883,372.602,-24.299,21.444,-41.938
C04470=1016.999,83.235,372.568,-24.300,21.444,-41.935
C04471=1016.997,83.586,372.534,-24.300,21.444,-41.931
C04472=1016.997,83.936,372.501,-24.301,21.443,-41.929
C04473=1016.995,84.284,372.467,-24.301,21.443,-41.925
C04474=1016.994,84.633,372.433,-24.302,21.443,-41.922
C04475=1016.993,84.979,372.400,-24.302,21.443,-41.918
C04476=1016.992,85.325,372.366,-24.302,21.442,-41.916
C04477=1016.990,85.669,372.334,-24.303,21.442,-41.912
C04478=1016.990,86.012,372.300,-24.303,21.442,-41.909
C04479=1016.988,86.354,372.267,-24.304,21.441,-41.906
C04480=1016.987,86.695,372.234,-24.304,21.441,-41.903
C04481=1016.986,87.034,372.201,-24.305,21.441,-41.899
C04482=1016.985,87.371,372.169,-24.305,21.441,-41.898
C04483=1016.983,87.703,372.137,-24.305,21.440,-41.894
C04484=1016.982,88.030,372.104,-24.306,21.441,-41.890
C04485=1016.981,88.352,372.073,-24.306,21.439,-41.888
C04486=1016.981,88.672,372.042,-24.307,21.440,-41.885
C04487=1016.979,88.994,372.011,-24.307,21.439,-41.881
C04488=1016.978,89.319,371.980,-24.308,21.439,-41.879
C04489=1016.976,89.648,371.948,-24.308,21.440,-41.876
C04490=1016.976,89.981,371.916,-24.308,21.438,-41.874
C04491=1016.975,90.315,371.883,-24.309,21.439,-41.870
C04492=1016.973,90.650,371.851,-24.309,21.438,-41.866
C04493=1016.972,90.984,371.819,-24.310,21.438,-41.865
C04494=1016.971,91.319,371.786,-24.310,21.438,-41.861
C04495=1016.970,91.653,371.753,-24.311,21.438,-41.857
C04496=1016.968,91.987,371.721,-24.311,21.437,-41.855
C04497=1016.967,92.322,371.688,-24.311,21.437,-41.852
C04498=1016.966,92.657,371.655,-24.312,21.436,-41.849
C04499=1016.966,92.990,371.623,-24.312,21.437,-41.846
C04500=1016.964,93.325,371.590,-24.313,21.436,-41.842
C04501=1016.963,93.659,371.558,-24.313,21.436,-41.841
C04502=1016.961,93.993,371.525,-24.314,21.436,-41.837
C04503=1016.960,94.328,371.492,-24.314,21.436,-41.833
C04504=1016.959,94.662,371.459,-24.314,21.436,-41.832
C04505=1016.958,94.996,371.427,-24.315,21.435,-41.828
C04506=1016.957,95.330,371.395,-24.315,21.435,-41.826
C04507=1016.955,95.665,371.362,-24.316,21.435,-41.822
C04508=1016.954,96.000,371.329,-24.316,21.435,-41.819
C04509=1016.953,96.334,371.296,-24.316,21.434,-41.817
C04510=1016.952,96.668,371.264,-24.317,21.434,-41.813
C04511=1016.950,97.002,371.231,-24.317,21.434,-41.811
C04512=1016.949,97.336,371.198,-24.318,21.434,-41.808
C04513=1016.948,97.670,371.166,-24.318,21.433,-41.806
C04514=1016.948,98.005,371.133,-24.318,21.433,-41.802
C04515=1016.946,98.339,371.100,-24.319,21.433,-41.799
C04516=1016.945,98.673,371.067,-24.319,21.432,-41.796
C04517=1016.943,99.007,371.035,-24.320,21.433,-41.793
C04518=1016.942,99.341,371.002,-24.320,21.432,-41.791
C04519=1016.941,99.676,370.969,-24.320,21.432,-41.787
C04520=1016.940,100.009,370.936,-24.321,21.432,-41.785
C04521=1016.939,100.344,370.903,-24.321,21.431,-41.782
C04522=1016.937,100.679,370.871,-24.322,21.432,-41.778
C04523=1016.936,101.012,370.837,-24.322,21.431,-41.776
C04524=1016.934,101.347,370.805,-24.323,21.431,-41.773
C04525=1016.933,101.680,370.772,-24.323,21.431,-41.771
C04526=1016.932,102.015,370.739,-24.323,21.430,-41.767
C04527=1016.931,102.348,370.706,-24.324,21.430,-41.765
C04528=1016.929,102.683,370.673,-24.324,21.431,-41.762
C04529=1016.929,103.016,370.641,-24.324,21.429,-41.760
C04530=1016.928,103.351,370.608,-24.325,21.430,-41.756
C04531=1016.927,103.685,370.575,-24.325,21.429,-41.752
C04532=1016.925,104.019,370.541,-24.326,21.429,-41.751
C04533=1016.924,104.353,370.509,-24.326,21.430,-41.747
C04534=1016.923,104.687,370.476,-24.326,21.428,-41.745
C04535=1016.921,105.021,370.443,-24.327,21.429,-41.742
C04536=1016.919,105.355,370.409,-24.327,21.428,-41.739
C04537=1016.918,105.689,370.376,-24.328,21.428,-41.736
C04538=1016.917,106.023,370.344,-24.328,21.428,-41.734
C04539=1016.916,106.357,370.310,-24.328,21.427,-41.730
C04540=1016.915,106.691,370.277,-24.329,21.427,-41.728
C04541=1016.914,107.026,370.244,-24.329,21.428,-41.725
C04542=1016.912,107.359,370.211,-24.329,21.427,-41.723
C04543=1016.911,107.693,370.178,-24.330,21.427,-41.719
C04544=1016.910,108.028,370.145,-24.330,21.427,-41.718
C04545=1016.908,108.361,370.112,-24.331,21.426,-41.714
C04546=1016.907,108.695,370.079,-24.331,21.426,-41.712
C04547=1016.906,109.029,370.046,-24.332,21.426,-41.708
C04548=1016.905,109.363,370.013,-24.332,21.425,-41.706
C04549=1016.903,109.697,369.980,-24.332,21.426,-41.703
C04550=1016.902,110.031,369.946,-24.333,21.425,-41.701
C04551=1016.901,110.366,369.913,-24.333,21.425,-41.697
C04552=1016.899,110.700,369.880,-24.333,21.425,-41.695
C04553=1016.898,111.033,369.847,-24.334,21.424,-41.692
C04554=1016.897,111.367,369.814,-24.334,21.424,-41.690
C04555=1016.896,111.701,369.780,-24.335,21.425,-41.686
C04556=1016.894,112.035,369.748,-24.335,21.423,-41.684
C04557=1016.893,112.369,369.714,-24.335,21.424,-41.681
C04558=1016.891,112.703,369.681,-24.336,21.424,-41.679
C04559=1016.891,113.037,369.647,-24.336,21.423,-41.675
C04560=1016.890,113.371,369.614,-24.336,21.423,-41.673
C04561=1016.888,113.705,369.581,-24.337,21.423,-41.670
C04562=1016.887,114.039,369.547,-24.337,21.422,-41.668
C04563=1016.885,114.373,369.515,-24.338,21.423,-41.664
C04564=1016.884,114.707,369.481,-24.338,21.422,-41.662
C04565=1016.883,115.040,369.448,-24.338,21.421,-41.660
C04566=1016.882,115.374,369.415,-24.339,21.422,-41.657
C04567=1016.880,115.709,369.381,-24.339,21.422,-41.655
C04568=1016.879,116.043,369.348,-24.340,21.422,-41.652
C04569=1016.878,116.376,369.314,-24.340,21.421,-41.649
C04570=1016.877,116.710,369.281,-24.340,21.421,-41.646
C04571=1016.875,117.044,369.247,-24.341,21.421,-41.644
C04572=1016.874,117.378,369.214,-24.341,21.421,-41.640
C04573=1016.873,117.712,369.180,-24.341,21.420,-41.638
C04574=1016.871,118.046,369.147,-24.342,21.421,-41.635
C04575=1016.870,118.380,369.113,-24.342,21.420,-41.633
C04576=1016.869,118.714,369.080,-24.342,21.419,-41.631
C04577=1016.867,119.048,369.046,-24.343,21.420,-41.628
C04578=1016.866,119.382,369.013,-24.343,21.419,-41.625
C04579=1016.865,119.716,368.980,-24.344,21.419,-41.622
C04580=1016.863,120.050,368.946,-24.344,21.419,-41.620
C04581=1016.862,120.384,368.913,-24.345,21.419,-41.617
C04582=1016.861,120.717,368.879,-24.345,21.418,-41.614
C04583=1016.859,121.051,368.846,-24.345,21.418,-41.613
C04584=1016.858,121.386,368.812,-24.346,21.418,-41.609
C04585=1016.857,121.720,368.779,-24.346,21.417,-41.607
C04586=1016.855,122.054,368.745,-24.346,21.418,-41.604
C04587=1016.854,122.387,368.712,-24.347,21.418,-41.602
C04588=1016.852,122.721,368.678,-24.347,21.418,-41.598
C04589=1016.851,123.056,368.644,-24.347,21.417,-41.596
C04590=1016.850,123.390,368.611,-24.348,21.417,-41.594
C04591=1016.849,123.723,368.577,-24.348,21.417,-41.591
C04592=1016.848,124.057,368.543,-24.348,21.417,-41.589
C04593=1016.846,124.391,368.509,-24.349,21.416,-41.585
C04594=1016.845,124.725,368.476,-24.349,21.416,-41.583
C04595=1016.843,125.059,368.442,-24.349,21.416,-41.581
C04596=1016.842,125.393,368.409,-24.350,21.416,-41.578
C04597=1016.841,125.728,368.375,-24.350,21.415,-41.576
C04598=1016.839,126.061,368.341,-24.351,21.416,-41.572
C04599=1016.838,126.395,368.307,-24.351,21.415,-41.571
C04600=1016.837,126.729,368.273,-24.351,21.415,-41.569
C04601=1016.835,127.063,368.240,-24.352,21.415,-41.565
C04602=1016.834,127.397,368.206,-24.352,21.415,-41.563
C04603=1016.833,127.732,368.172,-24.352,21.414,-41.561
C04604=1016.832,128.065,368.139,-24.353,21.415,-41.558
C04605=1016.830,128.399,368.104,-24.353,21.414,-41.555
C04606=1016.829,128.733,368.071,-24.354,21.414,-41.552
C04607=1016.828,129.067,368.037,-24.354,21.414,-41.550
C04608=1016.826,129.401,368.003,-24.354,21.414,-41.548
C04609=1016.825,129.736,367.970,-24.355,21.413,-41.545
C04610=1016.823,130.069,367.935,-24.355,21.413,-41.543
C04611=1016.823,130.404,367.901,-24.355,21.413,-41.541
C04612=1016.821,130.738,367.868,-24.356,21.413,-41.538
C04613=1016.819,131.072,367.834,-24.356,21.412,-41.535
C04614=1016.818,131.406,367.800,-24.356,21.412,-41.532
C04615=1016.817,131.739,367.766,-24.357,21.412,-41.530
C04616=1016.816,132.074,367.732,-24.357,21.412,-41.528
C04617=1016.814,132.408,367.698,-24.357,21.412,-41.525
C04618=1016.813,132.743,367.664,-24.358,21.411,-41.523
C04619=1016.811,133.076,367.630,-24.358,21.411,-41.521
C04620=1016.811,133.411,367.596,-24.358,21.411,-41.517
C04621=1016.809,133.745,367.562,-24.359,21.411,-41.515
C04622=1016.808,134.079,367.527,-24.359,21.410,-41.513
C04623=1016.807,134.412,367.494,-24.359,21.411,-41.510
C04624=1016.805,134.747,367.460,-24.360,21.410,-41.508
C04625=1016.804,135.081,367.426,-24.360,21.410,-41.506
C04626=1016.803,135.414,367.392,-24.361,21.411,-41.503
C04627=1016.801,135.737,367.359,-24.361,21.410,-41.501
C04628=1016.800,136.038,367.328,-24.361,21.410,-41.499
C04629=1016.799,136.317,367.299,-24.361,21.410,-41.497
C04630=1016.798,136.582,367.273,-24.361,21.409,-41.495
C04631=1016.796,136.846,367.246,-24.362,21.409,-41.491
C04632=1016.796,137.122,367.218,-24.362,21.409,-41.490
C04633=1016.795,137.420,367.187,-24.363,21.409,-41.488
C04634=1016.793,137.741,367.154,-24.363,21.408,-41.486
C04635=1016.791,138.082,367.119,-24.363,21.408,-41.484
C04636=1016.790,138.439,367.083,-24.364,21.408,-41.480
C04637=1016.789,138.850,367.041,-24.364,21.408,-41.477
C04638=1016.788,139.077,367.018,-24.364,21.408,-41.475
C04639=1016.787,139.316,366.993,-24.365,21.408,-41.473
C04640=1016.785,139.558,366.968,-24.365,21.408,-41.473
C04641=1016.785,139.798,366.944,-24.365,21.408,-41.471
C04642=1016.784,140.031,366.920,-24.365,21.408,-41.470
C04643=1016.783,140.252,366.897,-24.365,21.407,-41.469
C04644=1016.782,140.645,366.857,-24.366,21.407,-41.465
C04645=1016.780,140.989,366.822,-24.366,21.407,-41.462
C04646=1016.779,141.329,366.787,-24.367,21.407,-41.460
C04647=1016.778,141.668,366.752,-24.367,21.407,-41.457
C04648=1016.776,142.008,366.717,-24.367,21.406,-41.455
C04649=1016.776,142.349,366.682,-24.368,21.406,-41.453
C04650=1016.774,142.691,366.647,-24.368,21.407,-41.449
C04651=1016.772,143.033,366.612,-24.368,21.406,-41.448
C04652=1016.771,143.375,366.577,-24.369,21.405,-41.445
C04653=1016.770,143.718,366.541,-24.369,21.406,-41.442
C04654=1016.768,144.062,366.506,-24.369,21.405,-41.440
C04655=1016.767,144.406,366.471,-24.370,21.405,-41.438
C04656=1016.766,144.750,366.435,-24.370,21.406,-41.435
C04657=1016.765,145.096,366.400,-24.370,21.405,-41.432
C04658=1016.763,145.441,366.364,-24.371,21.404,-41.431
C04659=1016.762,145.787,366.328,-24.371,21.405,-41.427
C04660=1016.761,146.133,366.293,-24.371,21.405,-41.425
C04661=1016.759,146.478,366.257,-24.372,21.404,-41.424
C04662=1016.756,146.826,366.223,-24.372,21.404,-41.420
C04663=1016.740,147.171,366.195,-24.372,21.404,-41.418
C04664=1017.131,147.198,365.952,-24.372,21.404,-41.418
C04665=1017.148,146.853,365.978,-24.372,21.404,-41.420
C04666=1017.152,146.507,366.013,-24.372,21.404,-41.424
C04667=1017.153,146.161,366.048,-24.371,21.405,-41.425
C04668=1017.154,145.815,366.084,-24.371,21.405,-41.427
C04669=1017.156,145.469,366.119,-24.371,21.404,-41.431
C04670=1017.157,145.124,366.155,-24.370,21.405,-41.432
C04671=1017.158,144.779,366.190,-24.370,21.406,-41.435
C04672=1017.160,144.435,366.226,-24.370,21.405,-41.438
C04673=1017.161,144.090,366.262,-24.369,21.405,-41.440
C04674=1017.162,143.747,366.296,-24.369,21.406,-41.442
C04675=1017.164,143.403,366.333,-24.369,21.405,-41.445
C04676=1017.165,143.061,366.368,-24.368,21.406,-41.448
C04677=1017.166,142.719,366.403,-24.368,21.407,-41.449
C04678=1017.168,142.378,366.437,-24.368,21.406,-41.453
C04679=1017.169,142.037,366.473,-24.367,21.406,-41.455
C04680=1017.170,141.696,366.508,-24.367,21.407,-41.457
C04681=1017.171,141.357,366.543,-24.367,21.407,-41.460
C04682=1017.172,141.018,366.577,-24.366,21.407,-41.462
C04683=1017.174,140.673,366.613,-24.366,21.407,-41.465
C04684=1017.176,140.280,366.653,-24.365,21.407,-41.469
C04685=1017.176,140.060,366.675,-24.365,21.408,-41.470
C04686=1017.177,139.827,366.700,-24.365,21.408,-41.471
C04687=1017.178,139.586,366.724,-24.365,21.408,-41.473
C04688=1017.179,139.344,366.749,-24.365,21.408,-41.473
C04689=1017.180,139.107,366.773,-24.364,21.408,-41.475
C04690=1017.181,138.879,366.796,-24.364,21.408,-41.477
C04691=1017.183,138.468,366.839,-24.364,21.408,-41.480
C04692=1017.184,138.111,366.875,-24.363,21.408,-41.484
C04693=1017.185,137.771,366.910,-24.363,21.408,-41.486
C04694=1017.186,137.448,366.943,-24.363,21.409,-41.488
C04695=1017.188,137.150,366.973,-24.362,21.409,-41.490
C04696=1017.189,136.875,367.001,-24.362,21.409,-41.491
C04697=1017.190,136.611,367.028,-24.361,21.409,-41.495
C04698=1017.191,136.345,367.056,-24.361,21.410,-41.497
C04699=1017.192,136.066,367.084,-24.361,21.410,-41.499
C04700=1017.193,135.766,367.115,-24.361,21.410,-41.501
C04701=1017.195,135.443,367.147,-24.361,21.411,-41.503
C04702=1017.196,135.109,367.182,-24.360,21.410,-41.506
C04703=1017.197,134.775,367.215,-24.360,21.410,-41.508
C04704=1017.198,134.442,367.250,-24.359,21.411,-41.510
C04705=1017.200,134.107,367.284,-24.359,21.410,-41.513
C04706=1017.201,133.773,367.317,-24.359,21.411,-41.515
C04707=1017.202,133.438,367.351,-24.358,21.411,-41.517
C04708=1017.204,133.105,367.386,-24.358,21.411,-41.521
C04709=1017.204,132.770,367.419,-24.358,21.411,-41.523
C04710=1017.206,132.436,367.453,-24.357,21.412,-41.525
C04711=1017.207,132.102,367.488,-24.357,21.412,-41.528
C04712=1017.209,131.769,367.521,-24.357,21.412,-41.530
C04713=1017.210,131.434,367.556,-24.356,21.412,-41.532
C04714=1017.212,131.100,367.589,-24.356,21.412,-41.535
C04715=1017.213,130.766,367.623,-24.356,21.413,-41.538
C04716=1017.214,130.432,367.658,-24.355,21.413,-41.541
C04717=1017.216,130.098,367.691,-24.355,21.413,-41.543
C04718=1017.216,129.764,367.725,-24.355,21.413,-41.545
C04719=1017.218,129.429,367.759,-24.354,21.414,-41.548
C04720=1017.219,129.096,367.793,-24.354,21.414,-41.550
C04721=1017.221,128.762,367.827,-24.354,21.414,-41.552
C04722=1017.222,128.428,367.860,-24.353,21.414,-41.555
C04723=1017.223,128.093,367.894,-24.353,21.415,-41.558
C04724=1017.225,127.759,367.928,-24.352,21.414,-41.561
C04725=1017.226,127.426,367.962,-24.352,21.415,-41.563
C04726=1017.227,127.091,367.996,-24.352,21.415,-41.565
C04727=1017.228,126.758,368.029,-24.351,21.415,-41.569
C04728=1017.230,126.424,368.063,-24.351,21.415,-41.571
C04729=1017.231,126.089,368.097,-24.351,21.416,-41.572
C04730=1017.233,125.755,368.131,-24.350,21.415,-41.576
C04731=1017.234,125.422,368.165,-24.350,21.416,-41.578
C04732=1017.236,125.088,368.198,-24.349,21.416,-41.581
C04733=1017.236,124.754,368.232,-24.349,21.416,-41.583
C04734=1017.238,124.419,368.266,-24.349,21.416,-41.585
C04735=1017.239,124.086,368.299,-24.348,21.417,-41.589
C04736=1017.240,123.751,368.333,-24.348,21.417,-41.591
C04737=1017.242,123.417,368.366,-24.348,21.417,-41.594
C04738=1017.243,123.084,368.400,-24.347,21.417,-41.596
C04739=1017.245,122.750,368.434,-24.347,21.418,-41.598
C04740=1017.245,122.416,368.468,-24.347,21.418,-41.602
C04741=1017.246,122.082,368.501,-24.346,21.418,-41.604
C04742=1017.248,121.748,368.535,-24.346,21.417,-41.607
C04743=1017.249,121.414,368.568,-24.346,21.418,-41.609
C04744=1017.251,121.080,368.602,-24.345,21.418,-41.613
C04745=1017.252,120.746,368.635,-24.345,21.418,-41.614
C04746=1017.253,120.412,368.669,-24.345,21.419,-41.617
C04747=1017.255,120.078,368.702,-24.344,21.419,-41.620
C04748=1017.256,119.744,368.736,-24.344,21.419,-41.622
C04749=1017.257,119.410,368.769,-24.343,21.419,-41.625
C04750=1017.259,119.076,368.803,-24.343,21.420,-41.628
C04751=1017.260,118.742,368.836,-24.342,21.419,-41.631
C04752=1017.261,118.408,368.869,-24.342,21.420,-41.633
C04753=1017.263,118.074,368.903,-24.342,21.421,-41.635
C04754=1017.264,117.741,368.937,-24.341,21.420,-41.638
C04755=1017.265,117.406,368.970,-24.341,21.421,-41.640
C04756=1017.266,117.073,369.003,-24.341,21.421,-41.644
C04757=1017.268,116.739,369.037,-24.340,21.421,-41.646
C04758=1017.269,116.405,369.070,-24.340,21.421,-41.649
C04759=1017.270,116.071,369.104,-24.340,21.422,-41.652
C04760=1017.271,115.737,369.137,-24.339,21.422,-41.655
C04761=1017.273,115.403,369.171,-24.339,21.422,-41.657
C04762=1017.274,115.069,369.204,-24.338,21.421,-41.660
C04763=1017.275,114.735,369.237,-24.338,21.422,-41.662
C04764=1017.276,114.401,369.271,-24.338,21.423,-41.664
C04765=1017.278,114.067,369.304,-24.337,21.422,-41.668
C04766=1017.280,113.733,369.337,-24.337,21.423,-41.670
C04767=1017.281,113.399,369.370,-24.336,21.423,-41.673
C04768=1017.281,113.065,369.404,-24.336,21.423,-41.675
C04769=1017.282,112.731,369.437,-24.336,21.424,-41.679
C04770=1017.284,112.397,369.470,-24.335,21.424,-41.681
C04771=1017.286,112.063,369.504,-24.335,21.423,-41.684
C04772=1017.287,111.729,369.537,-24.335,21.425,-41.686
C04773=1017.288,111.395,369.570,-24.334,21.424,-41.690
C04774=1017.289,111.062,369.603,-24.334,21.424,-41.692
C04775=1017.291,110.728,369.636,-24.333,21.425,-41.695
C04776=1017.292,110.394,369.669,-24.333,21.425,-41.697
C04777=1017.293,110.059,369.702,-24.333,21.425,-41.701
C04778=1017.295,109.725,369.736,-24.332,21.426,-41.703
C04779=1017.296,109.391,369.769,-24.332,21.425,-41.706
C04780=1017.297,109.058,369.803,-24.332,21.426,-41.708
C04781=1017.298,108.723,369.835,-24.331,21.426,-41.712
C04782=1017.300,108.390,369.868,-24.331,21.426,-41.714
C04783=1017.301,108.056,369.901,-24.330,21.427,-41.718
C04784=1017.302,107.722,369.935,-24.330,21.427,-41.719
C04785=1017.303,107.388,369.967,-24.329,21.427,-41.723
C04786=1017.304,107.053,370.001,-24.329,21.428,-41.725
C04787=1017.305,106.720,370.034,-24.329,21.427,-41.728
C04788=1017.307,106.385,370.066,-24.328,21.427,-41.730
C04789=1017.308,106.052,370.100,-24.328,21.428,-41.734
C04790=1017.309,105.718,370.133,-24.328,21.428,-41.736
C04791=1017.311,105.384,370.165,-24.327,21.428,-41.739
C04792=1017.312,105.050,370.199,-24.327,21.429,-41.742
C04793=1017.314,104.715,370.232,-24.326,21.428,-41.745
C04794=1017.315,104.381,370.265,-24.326,21.430,-41.747
C04795=1017.316,104.047,370.299,-24.326,21.429,-41.751
C04796=1017.317,103.713,370.331,-24.325,21.429,-41.752
C04797=1017.318,103.379,370.364,-24.325,21.430,-41.756
C04798=1017.319,103.045,370.396,-24.324,21.429,-41.760
C04799=1017.320,102.711,370.429,-24.324,21.431,-41.762
C04800=1017.322,102.377,370.462,-24.324,21.430,-41.765
C04801=1017.323,102.043,370.495,-24.323,21.430,-41.767
C04802=1017.324,101.709,370.528,-24.323,21.431,-41.771
C04803=1017.325,101.374,370.561,-24.323,21.431,-41.773
C04804=1017.326,101.040,370.594,-24.322,21.431,-41.776
C04805=1017.328,100.706,370.627,-24.322,21.432,-41.778
C04806=1017.329,100.372,370.659,-24.321,21.431,-41.782
C04807=1017.330,100.038,370.693,-24.321,21.432,-41.785
C04808=1017.332,99.704,370.725,-24.320,21.432,-41.787
C04809=1017.333,99.370,370.758,-24.320,21.432,-41.791
C04810=1017.334,99.035,370.791,-24.320,21.433,-41.793
C04811=1017.335,98.701,370.824,-24.319,21.432,-41.796
C04812=1017.337,98.367,370.857,-24.319,21.433,-41.799
C04813=1017.338,98.033,370.889,-24.318,21.433,-41.802
C04814=1017.339,97.699,370.921,-24.318,21.433,-41.806
C04815=1017.340,97.365,370.955,-24.318,21.434,-41.808
C04816=1017.341,97.030,370.987,-24.317,21.434,-41.811
C04817=1017.342,96.696,371.020,-24.317,21.434,-41.813
C04818=1017.343,96.362,371.053,-24.316,21.434,-41.817
C04819=1017.345,96.028,371.086,-24.316,21.435,-41.819
C04820=1017.346,95.693,371.118,-24.316,21.435,-41.822
C04821=1017.348,95.359,371.151,-24.315,21.435,-41.826
C04822=1017.348,95.025,371.184,-24.315,21.435,-41.828
C04823=1017.349,94.690,371.216,-24.314,21.436,-41.832
C04824=1017.351,94.356,371.249,-24.314,21.436,-41.833
C04825=1017.352,94.022,371.281,-24.314,21.436,-41.837
C04826=1017.353,93.688,371.314,-24.313,21.436,-41.841
C04827=1017.354,93.353,371.347,-24.313,21.436,-41.842
C04828=1017.355,93.019,371.379,-24.312,21.437,-41.846
C04829=1017.357,92.685,371.412,-24.312,21.436,-41.849
C04830=1017.358,92.350,371.444,-24.311,21.437,-41.852
C04831=1017.359,92.015,371.477,-24.311,21.437,-41.855
C04832=1017.360,91.681,371.510,-24.311,21.438,-41.857
C04833=1017.362,91.346,371.542,-24.310,21.438,-41.861
C04834=1017.363,91.012,371.574,-24.310,21.438,-41.865
C04835=1017.364,90.677,371.607,-24.309,21.438,-41.866
C04836=1017.365,90.344,371.640,-24.309,21.439,-41.870
C04837=1017.366,90.009,371.673,-24.308,21.438,-41.874
C04838=1017.368,89.676,371.704,-24.308,21.440,-41.876
C04839=1017.368,89.346,371.737,-24.308,21.439,-41.879
C04840=1017.369,89.022,371.768,-24.307,21.439,-41.881
C04841=1017.371,88.701,371.799,-24.307,21.440,-41.885
C04842=1017.371,88.380,371.830,-24.306,21.439,-41.888
C04843=1017.373,88.058,371.861,-24.306,21.441,-41.890
C04844=1017.374,87.732,371.893,-24.305,21.440,-41.894
C04845=1017.375,87.399,371.925,-24.305,21.441,-41.898
C04846=1017.376,87.063,371.958,-24.305,21.441,-41.899
C04847=1017.377,86.723,371.991,-24.304,21.441,-41.903
C04848=1017.378,86.382,372.023,-24.304,21.441,-41.906
C04849=1017.380,86.040,372.057,-24.303,21.442,-41.909
C04850=1017.380,85.697,372.090,-24.303,21.442,-41.912
C04851=1017.382,85.353,372.124,-24.302,21.442,-41.916
C04852=1017.383,85.007,372.157,-24.302,21.443,-41.918
C04853=1017.384,84.661,372.191,-24.302,21.443,-41.922
C04854=1017.385,84.313,372.223,-24.301,21.443,-41.925
C04855=1017.386,83.964,372.257,-24.301,21.443,-41.929
C04856=1017.387,83.614,372.291,-24.300,21.444,-41.931
C04857=1017.389,83.263,372.325,-24.300,21.444,-41.935
C04858=1017.390,82.912,372.359,-24.299,21.444,-41.938
C04859=1017.391,82.559,372.392,-24.299,21.444,-41.942
C04860=1017.392,82.204,372.427,-24.298,21.444,-41.945
C04861=1017.393,81.850,372.461,-24.298,21.445,-41.947
C04862=1017.394,81.495,372.495,-24.298,21.446,-41.951
C04863=1017.395,81.139,372.529,-24.297,21.445,-41.955
C04864=1017.397,80.782,372.564,-24.297,21.446,-41.958
C04865=1017.399,80.425,372.597,-24.296,21.446,-41.962
C04866=1017.399,80.071,372.632,-24.296,21.446,-41.964
C04867=1017.401,79.720,372.665,-24.295,21.447,-41.968
C04868=1017.402,79.375,372.698,-24.295,21.446,-41.971
C04869=1017.402,79.035,372.731,-24.295,21.448,-41.973
C04870=1017.403,78.703,372.763,-24.294,21.447,-41.977
C04871=1017.405,78.375,372.794,-24.293,21.448,-41.980
C04872=1017.406,78.050,372.825,-24.293,21.448,-41.984
C04873=1017.407,77.727,372.856,-24.292,21.448,-41.987
C04874=1017.408,77.403,372.888,-24.292,21.449,-41.990
C04875=1017.409,77.077,372.918,-24.292,21.449,-41.994
C04876=1017.410,76.746,372.950,-24.291,21.449,-41.997
C04877=1017.411,76.411,372.982,-24.291,21.449,-42.001
C04878=1017.412,76.069,373.015,-24.290,21.449,-42.004
C04879=1017.413,75.719,373.048,-24.290,21.450,-42.006
C04880=1017.414,75.366,373.082,-24.289,21.450,-42.010
C04881=1017.415,75.008,373.116,-24.289,21.450,-42.013
C04882=1017.416,74.651,373.150,-24.288,21.451,-42.017
C04883=1017.418,74.294,373.184,-24.288,21.451,-42.019
C04884=1017.418,73.938,373.218,-24.288,21.451,-42.023
C04885=1017.420,73.585,373.252,-24.287,21.452,-42.027
C04886=1017.420,73.233,373.285,-24.286,21.451,-42.030
C04887=1017.422,72.884,373.318,-24.286,21.452,-42.034
C04888=1017.422,72.537,373.351,-24.285,21.452,-42.037
C04889=1017.424,72.190,373.384,-24.285,21.453,-42.041
C04890=1017.425,71.844,373.418,-24.285,21.453,-42.043
C04891=1017.426,71.499,373.450,-24.284,21.453,-42.047
C04892=1017.427,71.155,373.483,-24.284,21.454,-42.051
C04893=1017.429,70.810,373.515,-24.283,21.453,-42.054
C04894=1017.429,70.466,373.548,-24.283,21.454,-42.058
C04895=1017.430,70.121,373.581,-24.282,21.454,-42.061
C04896=1017.431,69.777,373.613,-24.282,21.455,-42.063
C04897=1017.432,69.433,373.646,-24.281,21.455,-42.067
C04898=1017.433,69.090,373.679,-24.281,21.456,-42.071
C04899=1017.434,68.747,373.711,-24.280,21.455,-42.074
C04900=1017.435,68.407,373.743,-24.280,21.456,-42.078
C04901=1017.436,68.066,373.775,-24.279,21.456,-42.082
C04902=1017.437,67.727,373.808,-24.279,21.456,-42.085
C04903=1017.438,67.389,373.839,-24.279,21.457,-42.087
C04904=1017.439,67.052,373.871,-24.278,21.457,-42.091
C04905=1017.439,66.715,373.903,-24.278,21.457,-42.094
C04906=1017.441,66.380,373.935,-24.277,21.457,-42.098
C04907=1017.441,66.046,373.966,-24.277,21.458,-42.102
C04908=1017.443,65.707,373.998,-24.276,21.457,-42.105
C04909=1017.444,65.352,374.032,-24.276,21.459,-42.108
C04910=1017.446,64.976,374.067,-24.275,21.458,-42.113
C04911=1017.446,64.581,374.104,-24.274,21.459,-42.116
C04912=1017.448,64.194,374.140,-24.274,21.459,-42.120
C04913=1017.448,63.837,374.174,-24.274,21.460,-42.124
C04914=1017.449,63.464,374.208,-24.273,21.460,-42.128
C04915=1017.452,63.246,374.228,-24.273,21.461,-42.130
C04916=1017.455,63.022,374.247,-24.272,21.460,-42.131
C04917=1017.461,62.626,374.282,-24.272,21.460,-42.135
C04918=1017.465,62.290,374.312,-24.271,21.461,-42.139
C04919=1017.469,61.955,374.340,-24.271,21.461,-42.142
C04920=1017.474,61.619,374.370,-24.270,21.462,-42.146
C04921=1017.478,61.285,374.399,-24.270,21.461,-42.149
C04922=1017.484,60.950,374.428,-24.269,21.462,-42.153
C04923=1017.487,60.615,374.457,-24.269,21.462,-42.157
C04924=1017.492,60.280,374.487,-24.268,21.462,-42.160
C04925=1017.496,59.945,374.516,-24.268,21.463,-42.163
C04926=1017.501,59.610,374.544,-24.268,21.464,-42.166
C04927=1017.505,59.275,374.575,-24.267,21.464,-42.170
C04928=1017.510,58.940,374.603,-24.267,21.464,-42.173
C04929=1017.514,58.605,374.632,-24.266,21.464,-42.177
C04930=1017.519,58.270,374.662,-24.266,21.465,-42.181
C04931=1017.522,57.935,374.691,-24.265,21.464,-42.184
C04932=1017.526,57.600,374.720,-24.264,21.465,-42.188
C04933=1017.531,57.265,374.748,-24.264,21.465,-42.192
C04934=1017.535,56.930,374.778,-24.264,21.466,-42.194
C04935=1017.540,56.595,374.807,-24.263,21.466,-42.197
C04936=1017.544,56.260,374.836,-24.263,21.466,-42.201
C04937=1017.548,55.925,374.865,-24.262,21.467,-42.205
C04938=1017.553,55.590,374.895,-24.262,21.467,-42.209
C04939=1017.557,55.255,374.923,-24.261,21.467,-42.212
C04940=1017.561,54.920,374.953,-24.261,21.467,-42.216
C04941=1017.565,54.585,374.982,-24.260,21.468,-42.220
C04942=1017.569,54.250,375.010,-24.260,21.468,-42.223
C04943=1017.573,53.915,375.039,-24.259,21.468,-42.227
C04944=1017.577,53.580,375.068,-24.259,21.468,-42.230
C04945=1017.581,53.245,375.097,-24.258,21.469,-42.234
C04946=1017.585,52.910,375.126,-24.258,21.469,-42.238
C04947=1017.590,52.575,375.156,-24.257,21.470,-42.240
C04948=1017.594,52.240,375.185,-24.257,21.470,-42.244
C04949=1017.598,51.904,375.214,-24.256,21.470,-42.247
C04950=1017.602,51.570,375.243,-24.256,21.471,-42.251
C04951=1017.606,51.235,375.272,-24.255,21.471,-42.254
C04952=1017.610,50.900,375.300,-24.255,21.471,-42.258
C04953=1017.614,50.565,375.329,-24.254,21.471,-42.262
C04954=1017.617,50.230,375.359,-24.254,21.472,-42.266
C04955=1017.622,49.895,375.387,-24.253,21.472,-42.269
C04956=1017.626,49.560,375.416,-24.253,21.472,-42.273
C04957=1017.629,49.225,375.446,-24.252,21.473,-42.277
C04958=1017.634,48.891,375.474,-24.252,21.473,-42.280
C04959=1017.638,48.555,375.503,-24.251,21.473,-42.284
C04960=1017.641,48.220,375.533,-24.251,21.473,-42.287
C04961=1017.645,47.886,375.561,-24.250,21.474,-42.291
C04962=1017.649,47.550,375.590,-24.250,21.474,-42.295
C04963=1017.653,47.216,375.619,-24.249,21.475,-42.299
C04964=1017.657,46.881,375.648,-24.249,21.475,-42.302
C04965=1017.660,46.546,375.676,-24.248,21.475,-42.306
C04966=1017.664,46.210,375.705,-24.248,21.475,-42.309
C04967=1017.668,45.876,375.735,-24.247,21.476,-42.313
C04968=1017.672,45.541,375.763,-24.247,21.476,-42.317
C04969=1017.675,45.206,375.791,-24.246,21.477,-42.321
C04970=1017.679,44.871,375.821,-24.246,21.477,-42.325
C04971=1017.684,44.536,375.850,-24.245,21.477,-42.328
C04972=1017.687,44.201,375.878,-24.245,21.477,-42.332
C04973=1017.690,43.866,375.908,-24.244,21.478,-42.335
C04974=1017.694,43.532,375.935,-24.244,21.478,-42.339
C04975=1017.698,43.196,375.964,-24.243,21.479,-42.343
C04976=1017.701,42.862,375.993,-24.243,21.479,-42.347
C04977=1017.705,42.527,376.022,-24.242,21.479,-42.350
C04978=1017.709,42.192,376.050,-24.242,21.479,-42.354
C04979=1017.712,41.857,376.080,-24.241,21.480,-42.357
C04980=1017.715,41.522,376.108,-24.241,21.480,-42.361
C04981=1017.720,41.187,376.137,-24.240,21.481,-42.365
C04982=1017.723,40.853,376.166,-24.240,21.481,-42.369
C04983=1017.727,40.518,376.195,-24.239,21.481,-42.372
C04984=1017.730,40.183,376.223,-24.239,21.481,-42.376
C04985=1017.733,39.849,376.252,-24.238,21.482,-42.380
C04986=1017.737,39.513,376.281,-24.238,21.482,-42.383
C04987=1017.741,39.179,376.309,-24.237,21.483,-42.387
C04988=1017.744,38.844,376.338,-24.237,21.483,-42.391
C04989=1017.748,38.509,376.366,-24.236,21.483,-42.395
C04990=1017.751,38.174,376.396,-24.236,21.483,-42.398
C04991=1017.754,37.840,376.423,-24.235,21.484,-42.402
C04992=1017.758,37.505,376.452,-24.235,21.484,-42.405
C04993=1017.761,37.170,376.481,-24.234,21.485,-42.409
C04994=1017.765,36.836,376.509,-24.234,21.485,-42.413
C04995=1017.768,36.501,376.538,-24.233,21.485,-42.418
C04996=1017.771,36.166,376.567,-24.232,21.485,-42.422
C04997=1017.775,35.832,376.595,-24.232,21.486,-42.426
C04998=1017.778,35.497,376.624,-24.231,21.485,-42.429
C04999=1017.782,35.162,376.653,-24.231,21.486,-42.433
C05000=1017.785,34.828,376.681,-24.230,21.486,-42.437
C05001=1017.788,34.493,376.710,-24.230,21.487,-42.440
C05002=1017.791,34.158,376.738,-24.229,21.487,-42.444
C05003=1017.795,33.824,376.767,-24.229,21.488,-42.448
C05004=1017.798,33.489,376.795,-24.228,21.488,-42.452
C05005=1017.801,33.154,376.824,-24.228,21.489,-42.455
C05006=1017.805,32.820,376.852,-24.227,21.489,-42.459
C05007=1017.808,32.485,376.881,-24.226,21.489,-42.464
C05008=1017.811,32.150,376.909,-24.226,21.489,-42.468
C05009=1017.815,31.816,376.937,-24.225,21.489,-42.471
C05010=1017.817,31.482,376.966,-24.225,21.490,-42.475
C05011=1017.820,31.147,376.994,-24.224,21.490,-42.479
C05012=1017.823,30.813,377.023,-24.224,21.491,-42.483
C05013=1017.826,30.478,377.051,-24.223,21.491,-42.486
C05014=1017.830,30.144,377.080,-24.223,21.492,-42.490
C05015=1017.833,29.809,377.108,-24.222,21.492,-42.494
C05016=1017.835,29.475,377.136,-24.222,21.493,-42.498
C05017=1017.839,29.140,377.164,-24.221,21.492,-42.503
C05018=1017.842,28.806,377.193,-24.221,21.493,-42.507
C05019=1017.844,28.471,377.221,-24.220,21.493,-42.510
C05020=1017.848,28.137,377.250,-24.220,21.494,-42.514
C05021=1017.851,27.802,377.278,-24.219,21.494,-42.518
C05022=1017.854,27.469,377.306,-24.219,21.495,-42.522
C05023=1017.857,27.133,377.334,-24.218,21.494,-42.525
C05024=1017.860,26.800,377.363,-24.217,21.494,-42.530
C05025=1017.863,26.465,377.391,-24.217,21.495,-42.534
C05026=1017.866,26.130,377.420,-24.216,21.495,-42.538
C05027=1017.869,25.796,377.447,-24.216,21.496,-42.541
C05028=1017.872,25.462,377.476,-24.215,21.496,-42.545
C05029=1017.875,25.128,377.503,-24.215,21.497,-42.549
C05030=1017.877,24.793,377.533,-24.214,21.497,-42.553
C05031=1017.880,24.459,377.560,-24.213,21.497,-42.558
C05032=1017.883,24.132,377.588,-24.213,21.498,-42.560
C05033=1017.885,23.838,377.613,-24.213,21.498,-42.562
C05034=1017.888,23.586,377.634,-24.212,21.498,-42.565
C05035=1017.891,23.179,377.669,-24.211,21.499,-42.573
C05036=1017.895,22.769,377.702,-24.210,21.499,-42.580
C05037=1017.896,22.516,377.724,-24.210,21.500,-42.582
C05038=1017.899,22.221,377.749,-24.210,21.501,-42.584
C05039=1017.901,21.898,377.776,-24.209,21.500,-42.588
C05040=1017.905,21.541,377.807,-24.209,21.501,-42.593
C05041=1017.906,21.333,377.823,-24.208,21.501,-42.597
C05042=1017.908,21.107,377.842,-24.208,21.502,-42.599
C05043=1017.910,20.864,377.863,-24.208,21.502,-42.601
C05044=1017.912,20.617,377.884,-24.207,21.502,-42.603
C05045=1017.914,20.370,377.904,-24.207,21.502,-42.604
C05046=1017.916,20.134,377.925,-24.207,21.502,-42.608
C05047=1017.919,19.716,377.960,-24.206,21.503,-42.613
C05048=1017.922,19.368,377.989,-24.205,21.502,-42.619
C05049=1017.925,19.036,378.017,-24.205,21.503,-42.622
C05050=1017.927,18.704,378.044,-24.204,21.503,-42.626
C05051=1017.930,18.373,378.072,-24.204,21.504,-42.630
C05052=1017.933,18.042,378.100,-24.203,21.504,-42.634
C05053=1017.935,17.712,378.128,-24.202,21.504,-42.639
C05054=1017.938,17.382,378.155,-24.202,21.505,-42.643
C05055=1017.940,17.053,378.183,-24.201,21.505,-42.646
C05056=1017.942,16.724,378.211,-24.201,21.506,-42.650
C05057=1017.945,16.396,378.238,-24.200,21.506,-42.654
C05058=1017.948,16.069,378.265,-24.200,21.507,-42.658
C05059=1017.950,15.742,378.293,-24.199,21.507,-42.663
C05060=1017.952,15.415,378.320,-24.199,21.507,-42.667
C05061=1017.955,15.089,378.347,-24.198,21.508,-42.670
C05062=1017.957,14.764,378.374,-24.198,21.508,-42.674
C05063=1017.960,14.439,378.401,-24.197,21.509,-42.678
C05064=1017.962,14.114,378.428,-24.197,21.509,-42.682
C05065=1017.964,13.790,378.455,-24.196,21.509,-42.687
C05066=1017.966,13.466,378.482,-24.195,21.509,-42.691
C05067=1017.969,13.142,378.510,-24.195,21.510,-42.694
C05068=1017.971,12.818,378.536,-24.194,21.510,-42.698
C05069=1017.973,12.495,378.563,-24.194,21.511,-42.702
C05070=1017.976,12.171,378.590,-24.193,21.511,-42.707
C05071=1017.978,11.848,378.617,-24.193,21.511,-42.711
C05072=1017.981,11.524,378.644,-24.192,21.512,-42.715
C05073=1017.982,11.202,378.671,-24.192,21.512,-42.718
C05074=1017.985,10.881,378.698,-24.191,21.513,-42.722
C05075=1017.987,10.562,378.724,-24.191,21.513,-42.726
C05076=1017.989,10.245,378.750,-24.190,21.514,-42.730
C05077=1017.991,9.930,378.777,-24.190,21.514,-42.733
C05078=1017.993,9.616,378.802,-24.189,21.514,-42.738
C05079=1017.996,9.301,378.829,-24.188,21.515,-42.742
C05080=1017.997,8.986,378.855,-24.188,21.515,-42.746
C05081=1017.999,8.669,378.880,-24.187,21.516,-42.750
C05082=1018.001,8.351,378.907,-24.186,21.515,-42.755
C05083=1018.004,8.030,378.934,-24.186,21.516,-42.759
C05084=1018.006,7.707,378.961,-24.186,21.516,-42.762
C05085=1018.008,7.381,378.988,-24.185,21.517,-42.766
C05086=1018.010,7.054,379.015,-24.185,21.517,-42.770
C05087=1018.012,6.726,379.041,-24.184,21.518,-42.774
C05088=1018.015,6.397,379.069,-24.183,21.518,-42.779
C05089=1018.016,6.067,379.096,-24.183,21.518,-42.783
C05090=1018.018,5.738,379.124,-24.182,21.519,-42.786
C05091=1018.020,5.407,379.150,-24.181,21.518,-42.792
C05092=1018.022,5.077,379.178,-24.181,21.519,-42.795
C05093=1018.024,4.745,379.206,-24.180,21.519,-42.799
C05094=1018.026,4.413,379.232,-24.180,21.521,-42.803
C05095=1018.028,4.084,379.260,-24.179,21.520,-42.807
C05096=1018.031,3.771,379.286,-24.179,21.521,-42.810
C05097=1018.032,3.481,379.309,-24.179,21.521,-42.814
C05098=1018.034,3.212,379.332,-24.178,21.522,-42.818
C05099=1018.036,2.950,379.354,-24.177,21.522,-42.823
C05100=1018.037,2.681,379.375,-24.177,21.522,-42.827
C05101=1018.039,2.393,379.399,-24.176,21.523,-42.831
C05102=1018.040,2.081,379.425,-24.176,21.523,-42.834
C05103=1018.042,1.750,379.452,-24.175,21.523,-42.838
C05104=1018.044,1.417,379.479,-24.175,21.524,-42.842
C05105=1018.046,1.083,379.507,-24.174,21.525,-42.846
C05106=1018.048,0.748,379.535,-24.173,21.525,-42.851
C05107=1018.050,0.412,379.562,-24.173,21.525,-42.855
C05108=1018.052,0.075,379.590,-24.172,21.526,-42.858
C05109=1018.054,-0.264,379.617,-24.172,21.526,-42.864
C05110=1018.055,-0.604,379.645,-24.171,21.526,-42.867
C05111=1018.057,-0.946,379.673,-24.170,21.527,-42.873
C05112=1018.059,-1.289,379.701,-24.170,21.527,-42.877
C05113=1018.061,-1.633,379.729,-24.169,21.528,-42.880
C05114=1018.063,-1.980,379.758,-24.169,21.528,-42.886
C05115=1018.064,-2.329,379.786,-24.168,21.529,-42.890
C05116=1018.066,-2.679,379.814,-24.167,21.529,-42.895
C05117=1018.069,-3.030,379.844,-24.167,21.529,-42.899
C05118=1018.070,-3.382,379.872,-24.166,21.529,-42.904
C05119=1018.072,-3.737,379.902,-24.166,21.531,-42.908
C05120=1018.073,-4.094,379.931,-24.165,21.530,-42.913
C05121=1018.075,-4.456,379.960,-24.164,21.531,-42.919
C05122=1018.077,-4.822,379.989,-24.164,21.532,-42.923
C05123=1018.079,-5.193,380.020,-24.163,21.532,-42.928
C05124=1018.081,-5.566,380.051,-24.163,21.533,-42.932
C05125=1018.082,-5.941,380.081,-24.162,21.533,-42.937
C05126=1018.085,-6.317,380.111,-24.161,21.533,-42.941
C05127=1018.086,-6.692,380.141,-24.160,21.534,-42.947
C05128=1018.088,-7.064,380.172,-24.160,21.534,-42.952
C05129=1018.090,-7.432,380.202,-24.159,21.535,-42.956
C05130=1018.091,-7.798,380.232,-24.158,21.535,-42.961
C05131=1018.093,-8.162,380.261,-24.158,21.536,-42.967
C05132=1018.095,-8.524,380.291,-24.157,21.536,-42.971
C05133=1018.096,-8.887,380.320,-24.156,21.536,-42.976
C05134=1018.098,-9.250,380.349,-24.156,21.537,-42.982
C05135=1018.099,-9.612,380.379,-24.155,21.538,-42.985
C05136=1018.101,-9.974,380.408,-24.154,21.538,-42.991
C05137=1018.102,-10.335,380.437,-24.154,21.539,-42.995
C05138=1018.103,-10.695,380.466,-24.153,21.539,-43.000
C05139=1018.105,-11.054,380.495,-24.152,21.539,-43.006
C05140=1018.107,-11.411,380.524,-24.152,21.540,-43.009
C05141=1018.108,-11.767,380.553,-24.151,21.540,-43.014
C05142=1018.109,-12.123,380.582,-24.151,21.541,-43.019
C05143=1018.111,-12.476,380.610,-24.150,21.541,-43.024
C05144=1018.113,-12.828,380.638,-24.149,21.542,-43.028
C05145=1018.114,-13.178,380.667,-24.149,21.542,-43.033
C05146=1018.115,-13.526,380.695,-24.148,21.543,-43.037
C05147=1018.117,-13.873,380.722,-24.147,21.543,-43.042
C05148=1018.118,-14.217,380.751,-24.147,21.544,-43.046
C05149=1018.119,-14.559,380.777,-24.146,21.544,-43.052
C05150=1018.120,-14.900,380.805,-24.146,21.544,-43.055
C05151=1018.121,-15.238,380.832,-24.145,21.545,-43.061
C05152=1018.123,-15.574,380.859,-24.145,21.546,-43.065
C05153=1018.124,-15.909,380.886,-24.144,21.546,-43.070
C05154=1018.125,-16.243,380.913,-24.143,21.546,-43.074
C05155=1018.126,-16.577,380.940,-24.142,21.547,-43.079
C05156=1018.127,-16.910,380.967,-24.142,21.547,-43.083
C05157=1018.129,-17.243,380.993,-24.141,21.547,-43.088
C05158=1018.129,-17.576,381.019,-24.141,21.548,-43.092
C05159=1018.131,-17.941,381.049,-24.140,21.549,-43.100
C05160=1018.131,-18.163,381.067,-24.139,21.548,-43.103
C05161=1018.132,-18.410,381.086,-24.139,21.549,-43.105
C05162=1018.133,-18.672,381.107,-24.139,21.550,-43.107
C05163=1018.134,-18.934,381.129,-24.139,21.550,-43.109
C05164=1018.135,-19.182,381.148,-24.138,21.550,-43.112
C05165=1018.136,-19.598,381.182,-24.137,21.550,-43.118
C05166=1018.137,-19.770,381.195,-24.137,21.551,-43.122
C05167=1018.137,-20.103,381.222,-24.136,21.551,-43.127
C05168=1018.139,-20.436,381.248,-24.136,21.552,-43.131
C05169=1018.140,-20.769,381.275,-24.135,21.553,-43.135
C05170=1018.140,-21.102,381.301,-24.134,21.552,-43.140
C05171=1018.142,-21.434,381.328,-24.134,21.553,-43.144
C05172=1018.142,-21.767,381.354,-24.133,21.554,-43.149
C05173=1018.143,-22.100,381.381,-24.133,21.554,-43.153
C05174=1018.144,-22.433,381.407,-24.132,21.554,-43.158
C05175=1018.146,-22.766,381.434,-24.131,21.556,-43.162
C05176=1018.146,-23.098,381.460,-24.131,21.555,-43.168
C05177=1018.147,-23.431,381.487,-24.130,21.556,-43.171
C05178=1018.148,-23.764,381.513,-24.129,21.556,-43.177
C05179=1018.149,-24.097,381.539,-24.129,21.557,-43.181
C05180=1018.150,-24.430,381.565,-24.128,21.557,-43.186
C05181=1018.150,-24.762,381.592,-24.128,21.558,-43.190
C05182=1018.151,-25.095,381.618,-24.127,21.558,-43.195
C05183=1018.152,-25.427,381.645,-24.126,21.559,-43.199
C05184=1018.152,-25.761,381.671,-24.126,21.559,-43.204
C05185=1018.153,-26.094,381.697,-24.125,21.559,-43.208
C05186=1018.154,-26.427,381.724,-24.124,21.560,-43.214
C05187=1018.155,-26.759,381.750,-24.124,21.560,-43.217
C05188=1018.155,-27.092,381.777,-24.123,21.560,-43.223
C05189=1018.156,-27.425,381.802,-24.123,21.562,-43.227
C05190=1018.157,-27.758,381.829,-24.122,21.562,-43.232
C05191=1018.158,-28.090,381.855,-24.121,21.562,-43.236
C05192=1018.158,-28.423,381.882,-24.120,21.562,-43.241
C05193=1018.159,-28.756,381.907,-24.120,21.563,-43.245
C05194=1018.160,-29.088,381.933,-24.119,21.563,-43.250
C05195=1018.160,-29.421,381.960,-24.119,21.564,-43.254
C05196=1018.161,-29.753,381.986,-24.118,21.565,-43.260
C05197=1018.161,-30.086,382.012,-24.118,21.565,-43.264
C05198=1018.162,-30.419,382.038,-24.117,21.565,-43.269
C05199=1018.162,-30.751,382.064,-24.116,21.566,-43.273
C05200=1018.162,-31.085,382.091,-24.116,21.566,-43.278
C05201=1018.163,-31.418,382.116,-24.115,21.567,-43.282
C05202=1018.164,-31.750,382.143,-24.114,21.567,-43.287
C05203=1018.164,-32.083,382.169,-24.114,21.568,-43.291
C05204=1018.165,-32.416,382.195,-24.113,21.568,-43.296
C05205=1018.165,-32.749,382.221,-24.113,21.569,-43.301
C05206=1018.166,-33.081,382.247,-24.112,21.569,-43.306
C05207=1018.166,-33.414,382.273,-24.111,21.570,-43.310
C05208=1018.167,-33.747,382.299,-24.111,21.570,-43.315
C05209=1018.168,-34.079,382.325,-24.110,21.571,-43.319
C05210=1018.168,-34.411,382.351,-24.109,21.571,-43.324
C05211=1018.168,-34.745,382.376,-24.109,21.572,-43.328
C05212=1018.169,-35.077,382.403,-24.108,21.572,-43.334
C05213=1018.169,-35.410,382.429,-24.108,21.573,-43.337
C05214=1018.169,-35.743,382.454,-24.107,21.573,-43.343
C05215=1018.169,-36.076,382.481,-24.107,21.574,-43.347
C05216=1018.170,-36.408,382.507,-24.106,21.574,-43.352
C05217=1018.170,-36.740,382.533,-24.105,21.574,-43.357
C05218=1018.171,-37.073,382.558,-24.105,21.575,-43.361
C05219=1018.171,-37.406,382.585,-24.104,21.575,-43.366
C05220=1018.171,-37.738,382.610,-24.103,21.576,-43.371
C05221=1018.172,-38.071,382.636,-24.102,21.576,-43.376
C05222=1018.171,-38.404,382.661,-24.102,21.577,-43.380
C05223=1018.172,-38.736,382.688,-24.101,21.577,-43.385
C05224=1018.173,-39.069,382.713,-24.101,21.578,-43.389
C05225=1018.172,-39.402,382.739,-24.100,21.578,-43.394
C05226=1018.172,-39.735,382.766,-24.100,21.579,-43.398
C05227=1018.172,-40.067,382.791,-24.099,21.579,-43.404
C05228=1018.172,-40.400,382.816,-24.098,21.580,-43.409
C05229=1018.173,-40.733,382.842,-24.098,21.580,-43.413
C05230=1018.173,-41.065,382.868,-24.097,21.580,-43.418
C05231=1018.173,-41.397,382.894,-24.096,21.582,-43.422
C05232=1018.173,-41.730,382.919,-24.096,21.582,-43.427
C05233=1018.173,-42.063,382.945,-24.095,21.582,-43.431
C05234=1018.174,-42.395,382.971,-24.094,21.583,-43.437
C05235=1018.174,-42.728,382.996,-24.094,21.583,-43.442
C05236=1018.173,-43.061,383.022,-24.093,21.583,-43.446
C05237=1018.173,-43.393,383.048,-24.092,21.584,-43.451
C05238=1018.174,-43.726,383.073,-24.092,21.585,-43.455
C05239=1018.173,-44.058,383.099,-24.091,21.585,-43.461
C05240=1018.173,-44.391,383.124,-24.091,21.586,-43.465
C05241=1018.173,-44.723,383.149,-24.090,21.586,-43.470
C05242=1018.174,-45.056,383.176,-24.089,21.586,-43.475
C05243=1018.174,-45.389,383.201,-24.089,21.587,-43.479
C05244=1018.174,-45.721,383.226,-24.088,21.588,-43.485
C05245=1018.173,-46.053,383.252,-24.088,21.588,-43.488
C05246=1018.173,-46.386,383.277,-24.087,21.588,-43.494
C05247=1018.173,-46.718,383.303,-24.086,21.590,-43.498
C05248=1018.173,-47.051,383.328,-24.086,21.589,-43.503
C05249=1018.172,-47.384,383.354,-24.085,21.589,-43.508
C05250=1018.172,-47.716,383.379,-24.084,21.591,-43.512
C05251=1018.172,-48.049,383.404,-24.083,21.591,-43.518
C05252=1018.172,-48.381,383.430,-24.083,21.592,-43.522
C05253=1018.172,-48.713,383.456,-24.082,21.592,-43.527
C05254=1018.172,-49.046,383.481,-24.081,21.592,-43.532
C05255=1018.172,-49.378,383.506,-24.081,21.593,-43.536
C05256=1018.172,-49.711,383.531,-24.080,21.593,-43.542
C05257=1018.171,-50.043,383.557,-24.080,21.595,-43.546
C05258=1018.171,-50.375,383.582,-24.079,21.594,-43.551
C05259=1018.171,-50.708,383.607,-24.079,21.595,-43.555
C05260=1018.170,-51.040,383.633,-24.078,21.596,-43.560
C05261=1018.170,-51.373,383.657,-24.077,21.596,-43.566
C05262=1018.169,-51.705,383.683,-24.077,21.597,-43.570
C05263=1018.169,-52.037,383.709,-24.076,21.597,-43.575
C05264=1018.169,-52.370,383.734,-24.075,21.597,-43.579
C05265=1018.168,-52.702,383.759,-24.075,21.598,-43.584
C05266=1018.168,-53.034,383.784,-24.074,21.598,-43.589
C05267=1018.167,-53.367,383.809,-24.074,21.600,-43.594
C05268=1018.167,-53.699,383.834,-24.073,21.599,-43.599
C05269=1018.166,-54.031,383.860,-24.072,21.600,-43.603
C05270=1018.166,-54.363,383.885,-24.072,21.601,-43.608
C05271=1018.166,-54.696,383.910,-24.071,21.601,-43.613
C05272=1018.165,-55.028,383.935,-24.070,21.602,-43.618
C05273=1018.165,-55.360,383.960,-24.070,21.602,-43.623
C05274=1018.164,-55.694,383.985,-24.069,21.603,-43.627
C05275=1018.164,-56.026,384.010,-24.068,21.603,-43.632
C05276=1018.164,-56.359,384.036,-24.068,21.603,-43.637
C05277=1018.163,-56.692,384.060,-24.067,21.605,-43.642
C05278=1018.162,-57.025,384.086,-24.066,21.604,-43.647
C05279=1018.161,-57.359,384.111,-24.066,21.605,-43.652
C05280=1018.161,-57.693,384.136,-24.065,21.606,-43.656
C05281=1018.160,-58.027,384.161,-24.064,21.606,-43.662
C05282=1018.160,-58.361,384.186,-24.064,21.607,-43.666
C05283=1018.159,-58.696,384.211,-24.063,21.607,-43.671
C05284=1018.158,-59.032,384.237,-24.062,21.608,-43.676
C05285=1018.158,-59.368,384.261,-24.062,21.608,-43.680
C05286=1018.157,-59.704,384.287,-24.061,21.609,-43.686
C05287=1018.156,-60.040,384.312,-24.060,21.609,-43.691
C05288=1018.155,-60.377,384.337,-24.060,21.610,-43.695
C05289=1018.155,-60.714,384.363,-24.059,21.610,-43.700
C05290=1018.154,-61.052,384.388,-24.059,21.611,-43.706
C05291=1018.154,-61.390,384.413,-24.058,21.611,-43.710
C05292=1018.153,-61.728,384.438,-24.057,21.612,-43.715
C05293=1018.152,-62.067,384.464,-24.057,21.612,-43.720
C05294=1018.152,-62.406,384.489,-24.056,21.614,-43.725
C05295=1018.150,-62.746,384.515,-24.055,21.613,-43.730
C05296=1018.149,-63.086,384.540,-24.055,21.614,-43.735
C05297=1018.148,-63.426,384.565,-24.054,21.615,-43.739
C05298=1018.148,-63.767,384.590,-24.053,21.616,-43.745
C05299=1018.146,-64.108,384.616,-24.053,21.615,-43.750
C05300=1018.146,-64.449,384.641,-24.052,21.617,-43.754
C05301=1018.145,-64.791,384.667,-24.051,21.617,-43.759
C05302=1018.144,-65.132,384.692,-24.051,21.618,-43.765
C05303=1018.143,-65.475,384.717,-24.050,21.617,-43.770
C05304=1018.142,-65.817,384.743,-24.050,21.619,-43.774
C05305=1018.142,-66.160,384.768,-24.049,21.619,-43.780
C05306=1018.140,-66.502,384.794,-24.048,21.620,-43.785
C05307=1018.139,-66.845,384.819,-24.048,21.620,-43.789
C05308=1018.138,-67.188,384.844,-24.047,21.621,-43.795
C05309=1018.137,-67.532,384.870,-24.046,21.621,-43.800
C05310=1018.136,-67.875,384.895,-24.045,21.622,-43.805
C05311=1018.135,-68.219,384.921,-24.045,21.622,-43.809
C05312=1018.134,-68.563,384.946,-24.044,21.623,-43.815
C05313=1018.132,-68.906,384.972,-24.043,21.623,-43.820
C05314=1018.131,-69.250,384.997,-24.043,21.624,-43.824
C05315=1018.130,-69.595,385.022,-24.042,21.624,-43.829
C05316=1018.129,-69.938,385.048,-24.041,21.625,-43.835
C05317=1018.128,-70.282,385.074,-24.041,21.625,-43.840
C05318=1018.127,-70.626,385.099,-24.040,21.626,-43.844
C05319=1018.125,-70.970,385.124,-24.040,21.627,-43.850
C05320=1018.124,-71.315,385.149,-24.039,21.627,-43.855
C05321=1018.123,-71.659,385.175,-24.038,21.628,-43.861
C05322=1018.122,-72.003,385.200,-24.038,21.628,-43.865
C05323=1018.120,-72.347,385.225,-24.037,21.629,-43.870
C05324=1018.119,-72.691,385.251,-24.036,21.629,-43.875
C05325=1018.118,-73.034,385.276,-24.035,21.630,-43.881
C05326=1018.116,-73.378,385.301,-24.035,21.630,-43.885
C05327=1018.115,-73.722,385.326,-24.034,21.631,-43.890
C05328=1018.113,-74.066,385.351,-24.033,21.632,-43.896
C05329=1018.112,-74.409,385.377,-24.033,21.632,-43.901
C05330=1018.110,-74.753,385.402,-24.032,21.633,-43.905
C05331=1018.109,-75.096,385.427,-24.031,21.633,-43.911
C05332=1018.107,-75.439,385.452,-24.031,21.634,-43.916
C05333=1018.106,-75.782,385.477,-24.030,21.634,-43.920
C05334=1018.105,-76.125,385.502,-24.030,21.635,-43.926
C05335=1018.104,-76.468,385.527,-24.029,21.635,-43.931
C05336=1018.101,-76.810,385.552,-24.028,21.636,-43.936
C05337=1018.100,-77.152,385.576,-24.028,21.636,-43.940
C05338=1018.099,-77.495,385.602,-24.027,21.637,-43.946
C05339=1018.097,-77.836,385.626,-24.026,21.637,-43.951
C05340=1018.096,-78.178,385.652,-24.026,21.639,-43.955
C05341=1018.094,-78.519,385.676,-24.025,21.638,-43.960
C05342=1018.092,-78.860,385.701,-24.024,21.639,-43.966
C05343=1018.090,-79.200,385.726,-24.023,21.639,-43.971
C05344=1018.089,-79.540,385.751,-24.023,21.641,-43.975
C05345=1018.087,-79.880,385.775,-24.022,21.641,-43.981
C05346=1018.085,-80.219,385.800,-24.021,21.641,-43.986
C05347=1018.084,-80.559,385.824,-24.021,21.643,-43.990
C05348=1018.082,-80.897,385.849,-24.020,21.643,-43.995
C05349=1018.080,-81.236,385.873,-24.020,21.643,-44.001
C05350=1018.079,-81.573,385.897,-24.019,21.644,-44.005
C05351=1018.077,-81.910,385.922,-24.018,21.645,-44.010
C05352=1018.075,-82.248,385.946,-24.018,21.645,-44.016
C05353=1018.074,-82.584,385.971,-24.017,21.645,-44.021
C05354=1018.072,-82.920,385.995,-24.016,21.646,-44.025
C05355=1018.070,-83.256,386.019,-24.016,21.647,-44.031
C05356=1018.068,-83.591,386.043,-24.015,21.647,-44.036
C05357=1018.067,-83.925,386.068,-24.015,21.648,-44.040
C05358=1018.064,-84.260,386.092,-24.014,21.648,-44.045
C05359=1018.063,-84.609,386.117,-24.013,21.649,-44.051
C05360=1018.060,-85.007,386.146,-24.012,21.650,-44.056
C05361=1018.059,-85.219,386.160,-24.012,21.649,-44.060
C05362=1018.058,-85.433,386.176,-24.012,21.649,-44.062
C05363=1018.056,-85.842,386.205,-24.011,21.650,-44.067
C05364=1018.054,-86.201,386.231,-24.010,21.651,-44.073
C05365=1018.052,-86.530,386.255,-24.009,21.652,-44.078
C05366=1018.050,-86.853,386.278,-24.009,21.652,-44.082
C05367=1018.048,-87.169,386.301,-24.008,21.653,-44.088
C05368=1018.046,-87.481,386.323,-24.007,21.653,-44.093
C05369=1018.044,-87.792,386.345,-24.007,21.654,-44.097
C05370=1018.043,-88.105,386.367,-24.006,21.654,-44.102
C05371=1018.041,-88.423,386.390,-24.006,21.655,-44.106
C05372=1018.039,-88.794,386.417,-24.005,21.656,-44.114
C05373=1018.037,-89.014,386.432,-24.004,21.656,-44.117
C05374=1018.036,-89.247,386.449,-24.004,21.656,-44.119
C05375=1018.034,-89.485,386.466,-24.004,21.656,-44.121
C05376=1018.033,-89.717,386.482,-24.004,21.657,-44.123
C05377=1018.031,-90.122,386.512,-24.003,21.658,-44.130
C05378=1018.028,-90.460,386.536,-24.002,21.658,-44.136
C05379=1018.025,-90.790,386.559,-24.001,21.659,-44.141
C05380=1018.024,-91.120,386.582,-24.001,21.660,-44.145
C05381=1018.021,-91.448,386.606,-24.000,21.660,-44.150
C05382=1018.020,-91.776,386.629,-23.999,21.660,-44.156
C05383=1018.018,-92.104,386.653,-23.999,21.661,-44.160
C05384=1018.015,-92.431,386.676,-23.998,21.662,-44.165
C05385=1018.013,-92.758,386.699,-23.998,21.662,-44.169
C05386=1018.011,-93.084,386.722,-23.997,21.663,-44.175
C05387=1018.009,-93.410,386.745,-23.996,21.663,-44.180
C05388=1018.006,-93.735,386.768,-23.996,21.664,-44.184
C05389=1018.004,-94.060,386.792,-23.995,21.664,-44.189
C05390=1018.002,-94.383,386.814,-23.994,21.665,-44.193
C05391=1017.999,-94.707,386.837,-23.994,21.666,-44.199
C05392=1017.997,-95.030,386.860,-23.993,21.666,-44.204
C05393=1017.995,-95.352,386.883,-23.993,21.666,-44.207
C05394=1017.992,-95.676,386.905,-23.992,21.667,-44.213
C05395=1017.991,-95.997,386.928,-23.991,21.668,-44.217
C05396=1017.988,-96.318,386.951,-23.991,21.668,-44.222
C05397=1017.985,-96.640,386.974,-23.990,21.669,-44.226
C05398=1017.984,-96.962,386.997,-23.989,21.669,-44.231
C05399=1017.981,-97.282,387.019,-23.989,21.670,-44.236
C05400=1017.979,-97.603,387.042,-23.988,21.670,-44.241
C05401=1017.976,-97.924,387.064,-23.987,21.670,-44.246
C05402=1017.974,-98.245,387.087,-23.987,21.672,-44.250
C05403=1017.972,-98.566,387.110,-23.986,21.671,-44.255
C05404=1017.969,-98.887,387.132,-23.986,21.673,-44.260
C05405=1017.967,-99.208,387.155,-23.985,21.673,-44.265
C05406=1017.964,-99.529,387.177,-23.985,21.673,-44.268
C05407=1017.962,-99.851,387.200,-23.984,21.674,-44.274
C05408=1017.959,-100.173,387.222,-23.983,21.675,-44.278
C05409=1017.956,-100.495,387.245,-23.983,21.675,-44.283
C05410=1017.954,-100.818,387.268,-23.982,21.676,-44.287
C05411=1017.951,-101.140,387.290,-23.981,21.676,-44.292
C05412=1017.948,-101.464,387.313,-23.981,21.677,-44.298
C05413=1017.946,-101.789,387.335,-23.980,21.677,-44.302
C05414=1017.943,-102.113,387.358,-23.980,21.678,-44.307
C05415=1017.941,-102.438,387.381,-23.979,21.679,-44.311
C05416=1017.938,-102.763,387.404,-23.978,21.679,-44.316
C05417=1017.935,-103.090,387.426,-23.978,21.680,-44.320
C05418=1017.932,-103.415,387.449,-23.977,21.680,-44.326
C05419=1017.930,-103.743,387.472,-23.976,21.681,-44.331
C05420=1017.927,-104.070,387.494,-23.976,21.681,-44.335
C05421=1017.924,-104.398,387.517,-23.975,21.681,-44.340
C05422=1017.921,-104.726,387.540,-23.975,21.683,-44.344
C05423=1017.918,-105.054,387.564,-23.974,21.683,-44.350
C05424=1017.916,-105.383,387.587,-23.974,21.684,-44.354
C05425=1017.913,-105.712,387.610,-23.973,21.684,-44.359
C05426=1017.910,-106.041,387.632,-23.972,21.685,-44.365
C05427=1017.907,-106.369,387.654,-23.972,21.685,-44.368
C05428=1017.905,-106.698,387.678,-23.971,21.685,-44.374
C05429=1017.901,-107.028,387.701,-23.971,21.687,-44.378
C05430=1017.898,-107.356,387.723,-23.970,21.687,-44.383
C05431=1017.896,-107.686,387.746,-23.969,21.687,-44.388
C05432=1017.893,-108.014,387.769,-23.969,21.688,-44.392
C05433=1017.889,-108.343,387.792,-23.968,21.689,-44.398
C05434=1017.886,-108.672,387.814,-23.967,21.689,-44.402
C05435=1017.883,-109.001,387.837,-23.967,21.689,-44.407
C05436=1017.880,-109.330,387.860,-23.966,21.690,-44.412
C05437=1017.878,-109.659,387.883,-23.965,21.691,-44.416
C05438=1017.875,-109.988,387.905,-23.965,21.691,-44.422
C05439=1017.872,-110.317,387.928,-23.964,21.692,-44.426
C05440=1017.868,-110.646,387.951,-23.963,21.692,-44.431
C05441=1017.865,-110.974,387.974,-23.963,21.693,-44.436
C05442=1017.862,-111.303,387.997,-23.962,21.693,-44.440
C05443=1017.859,-111.632,388.019,-23.962,21.694,-44.446
C05444=1017.856,-111.961,388.041,-23.961,21.695,-44.449
C05445=1017.852,-112.290,388.064,-23.960,21.695,-44.455
C05446=1017.849,-112.618,388.086,-23.960,21.696,-44.459
C05447=1017.846,-112.947,388.109,-23.959,21.696,-44.464
C05448=1017.843,-113.275,388.132,-23.958,21.697,-44.470
C05449=1017.840,-113.604,388.154,-23.958,21.697,-44.473
C05450=1017.836,-113.932,388.177,-23.957,21.698,-44.479
C05451=1017.833,-114.261,388.199,-23.957,21.699,-44.483
C05452=1017.829,-114.590,388.222,-23.956,21.699,-44.488
C05453=1017.825,-114.918,388.244,-23.956,21.700,-44.492
C05454=1017.822,-115.247,388.267,-23.955,21.700,-44.497
C05455=1017.819,-115.575,388.290,-23.954,21.701,-44.503
C05456=1017.815,-115.904,388.312,-23.954,21.701,-44.507
C05457=1017.812,-116.232,388.335,-23.953,21.701,-44.512
C05458=1017.809,-116.561,388.357,-23.953,21.703,-44.516
C05459=1017.806,-116.889,388.379,-23.952,21.703,-44.521
C05460=1017.802,-117.217,388.402,-23.951,21.704,-44.525
C05461=1017.799,-117.546,388.424,-23.951,21.704,-44.531
C05462=1017.794,-117.875,388.447,-23.950,21.705,-44.535
C05463=1017.791,-118.203,388.469,-23.949,21.705,-44.540
C05464=1017.788,-118.532,388.491,-23.949,21.705,-44.545
C05465=1017.785,-118.860,388.514,-23.948,21.707,-44.549
C05466=1017.781,-119.189,388.536,-23.948,21.707,-44.554
C05467=1017.777,-119.517,388.558,-23.947,21.707,-44.558
C05468=1017.774,-119.845,388.581,-23.946,21.708,-44.564
C05469=1017.770,-120.174,388.603,-23.946,21.709,-44.568
C05470=1017.766,-120.502,388.625,-23.945,21.709,-44.573
C05471=1017.763,-120.830,388.647,-23.945,21.710,-44.577
C05472=1017.759,-121.158,388.671,-23.944,21.710,-44.582
C05473=1017.756,-121.486,388.693,-23.944,21.711,-44.586
